(* IEC 61131-3 sources: std_i2980_v2.06_cp053/Source/IMM/ieccontrol/GlobalBaseArchives (part 2) *)

(* ---- ABVersionManager.pu ---- *)
(*
This algorithm block contains algorithms for version reading:
IEC and HMI version from version info text file
Firmware version from catalog
and stores them to sv_HMIVersion, sv_IECVersion and sv_FirmwareVersion
*)

IMPORT_OVER_LISTFILE
 KCAT_GetHandle
, KFILE_Open
, KFILE_Close
, tsTraceLevel
, KCAT_HandleData
, KCAT_Status
, KCAT_GenericDataFlags
, KCAT_RetCode

END_IMPORT

ALGORITHM_BLOCK ABVersionManager #DUMMY_EDIT_BLOCK

SYSTEM_VAR
 sv_TraceLevel : tsTraceLevel;
END_VAR

VAR
 msOsVersion : STRING(255);
 msDeviceSwVersion : STRING(255);
 msFirmwareVersion : STRING(255);
 msSystemName : STRING(255);
 msIECVersion : STRING(255);
 msCustVersion : STRING(255);
 msKVBVersion : STRING(255);
 msLIBIECBase : STRING(255);
 msLIBIECLib : STRING(255);
 msLIBException : STRING(255);
 msLIBODC : STRING(255);
END_VAR

FUNCTION fHasVersionInfoExtended : BOOL
 #DUMMY_EDIT_BLOCK
#BEGIN_EDIT_BLOCK

fHasVersionInfoExtended := (msDeviceSwVersion <> 'no version info' AND msOsVersion <> 'no version info');

;#END_EDIT_BLOCK END_FUNCTION

(*
This algo will copy the firmware version from the catalog entry to the sv_FirmwareVersion
*)

ALGORITHM aReadVersionInfo

VAR_INPUT
 sNodeName : STRING(255);
END_VAR

VAR_IN_OUT
 sVersionInfo : STRING(255);
END_VAR

VAR
 DataHandle : KCAT_HandleData;
 KCATStatus : KCAT_Status;
 dummy : DINT;
END_VAR
#BEGIN_EDIT_BLOCK
DataHandle := KCAT_GetHandle(sNodeName);
KCATStatus := DataHandle.Status;

IF (KCATStatus = KCAT_Status_OK) THEN
   KCATStatus := KCAT_GetValue(DataHandle.Handle, sVersionInfo);
END_IF;

IF ((KCATStatus <> KCAT_Status_OK) OR (sVersionInfo = '')) THEN
   sVersionInfo := "no version info";
   dummy := Print('Entry %s could not be found in catalog', sNodeName);
END_IF;

;#END_EDIT_BLOCK END_ALGORITHM

(*
This algo will copy the firmware version from the catalog entry to the sv_FirmwareVersion
*)

ALGORITHM aReadAllVersionInfos

VAR
 dummy : DINT;
END_VAR
#BEGIN_EDIT_BLOCK
aReadVersionInfo('System.firmwareVersion', msFirmwareVersion);
aReadVersionInfo('Application.KePlast.systemName', msSystemName);
aReadVersionInfo('Application.KePlast.IEC.componentVersionString', msIECVersion);
aReadVersionInfo('Application.KePlast.HMI.KVB.componentVersionString', msKVBVersion);

//aReadVersionInfo('Application.ApplMoldMachineKVBBase.componentVersionString', msLIBKVBBase);
aReadVersionInfo('Application.ApplIECUserExceptionHandling.componentVersionString', msLIBException);
aReadVersionInfo('Application.ApplMoldMachineIECLib.componentVersionString', msLIBIECLib);
aReadVersionInfo('Application.ApplMoldMachineIECBase.componentVersionString', msLIBIECBase);
aReadVersionInfo('Application.ApplMoldMachineODC.componentVersionString', msLIBODC);
aReadVersionInfo('BootVis.displayText', msCustVersion);
aReadVersionInfo('System.OS.driversVersion', msDeviceSwVersion);
aReadVersionInfo('System.OS.osVersion', msOsVersion);

IF (sv_TraceLevel.bApplication) THEN
   dummy := Print('ABVersionManager.aReadAllVersionInfos:');
   dummy := Print('  Version System:   "%s"', msSystemName);
   dummy := Print('  Version Firmware: "%s"', msFirmwareVersion);
   dummy := Print('  Version IEC:      "%s"', msIECVersion);
   dummy := Print('  Version KVB:      "%s"', msKVBVersion);
   dummy := Print('  Version IECLib:   "%s"', msLIBIECLib);
   dummy := Print('  Version IECBase:  "%s"', msLIBIECBase);
   dummy := Print('  Version Customer: "%s"', msCustVersion);
   IF (fHasVersionInfoExtended()) THEN
      dummy := Print('  Version DeviceSw: "%s"', msDeviceSwVersion);
      dummy := Print('  Version OS:       "%s"', msOsVersion);
   END_IF;
   dummy := Print('--------------------------------------');
END_IF;

;#END_EDIT_BLOCK END_ALGORITHM

FUNCTION fGetSystemName : STRING(255)
 #DUMMY_EDIT_BLOCK
#BEGIN_EDIT_BLOCK
fGetSystemName := msSystemName;

;#END_EDIT_BLOCK END_FUNCTION

FUNCTION fGetIECVersion : STRING(255)
 #DUMMY_EDIT_BLOCK
#BEGIN_EDIT_BLOCK
fGetIECVersion := msIECVersion;

;#END_EDIT_BLOCK END_FUNCTION

FUNCTION fGetCustVersion : STRING(255)
 #DUMMY_EDIT_BLOCK
#BEGIN_EDIT_BLOCK
fGetCustVersion := msCustVersion;

;#END_EDIT_BLOCK END_FUNCTION

FUNCTION fGetLIBVersionIECBase : STRING(255)
 #DUMMY_EDIT_BLOCK
#BEGIN_EDIT_BLOCK
fGetLIBVersionIECBase := msLIBIECBase;

;#END_EDIT_BLOCK END_FUNCTION

FUNCTION fGetLIBVersionIECLib : STRING(255)
 #DUMMY_EDIT_BLOCK
#BEGIN_EDIT_BLOCK
fGetLIBVersionIECLib := msLIBIECLib;

;#END_EDIT_BLOCK END_FUNCTION

FUNCTION fGetLIBVersionIECException : STRING(255)
 #DUMMY_EDIT_BLOCK
#BEGIN_EDIT_BLOCK
fGetLIBVersionIECException := msLIBException;

;#END_EDIT_BLOCK END_FUNCTION

FUNCTION fGetKVBVersion : STRING(255)
 #DUMMY_EDIT_BLOCK
#BEGIN_EDIT_BLOCK
fGetKVBVersion := msKVBVersion;

;#END_EDIT_BLOCK END_FUNCTION

(*
read KVS version on each function call because it never will be available at startup of IEC
*)

FUNCTION fReadKVSVersion : STRING(255)
 #DUMMY_EDIT_BLOCK

VAR
 sKVSVersion : STRING(255);
END_VAR
#BEGIN_EDIT_BLOCK
aReadVersionInfo('Application.KePlast.HMI.KVS.componentVersionString', sKVSVersion);
fReadKVSVersion := sKVSVersion;

;#END_EDIT_BLOCK END_FUNCTION

FUNCTION fGetFirmwareVersion : STRING(255)
 #DUMMY_EDIT_BLOCK
#BEGIN_EDIT_BLOCK
fGetFirmwareVersion := msFirmwareVersion;

;#END_EDIT_BLOCK END_FUNCTION

FUNCTION fGetLIBVersionODC : STRING(255)
 #DUMMY_EDIT_BLOCK
#BEGIN_EDIT_BLOCK
fGetLIBVersionODC := msLIBODC;

;#END_EDIT_BLOCK END_FUNCTION

FUNCTION fGetCPUSerial : LINT
 #DUMMY_EDIT_BLOCK

VAR
 sSerialNumber : STRING(255);
 flags : KCAT_GenericDataFlags;
 catRetCode : KCAT_RetCode;
 catHdl : KCAT_HandleData;
END_VAR
#BEGIN_EDIT_BLOCK
// get cpu serial number
catHdl := KCAT_GetHandle('IO.ONBOARD');
IF (catHdl.Status = KCAT_Status_OK) THEN
   catRetCode := KCAT_GetGenericData(catHdl.Handle, KCAT_GDSelector_SerialNumber, flags, sSerialNumber);
   IF (catRetCode = 0) THEN
      fGetCPUSerial := STRING_TO_LINT(sSerialNumber);
   END_IF;
END_IF;

;#END_EDIT_BLOCK END_FUNCTION

FUNCTION fGetDeviceSoftwareVersion : STRING(255)
 #DUMMY_EDIT_BLOCK
#BEGIN_EDIT_BLOCK
fGetDeviceSoftwareVersion := msDeviceSwVersion;

;#END_EDIT_BLOCK END_FUNCTION

FUNCTION fGetOSVersion : STRING(255)
 #DUMMY_EDIT_BLOCK
#BEGIN_EDIT_BLOCK
fGetOSVersion := msOsVersion;

;#END_EDIT_BLOCK END_FUNCTION

END_ALGORITHM_BLOCK

#END_OF_IEC_PART

@Puma @IecEditor 6 97 @Pou 25
@@@BEG_Comment@@@
This algorithm block contains algorithms for version reading:
IEC and HMI version from version info text file
Firmware version from catalog
and stores them to sv_HMIVersion, sv_IECVersion and sv_FirmwareVersion
@@@END_Comment@@@

@BEG_Contents

@BEG_Func
@RT(17)FuncTreeContainer
3
@Var @RT(14)KCAT_GetHandle @RT(0) @T @T @DERIVED 0 @F @RT(22)KEBA_STANDARD_FUNCTION @F
@T
@BEG_Attrib
0 @RT(0) @RT(0)
@END_Attrib
1 1 @F @F @F @F

@Var @RT(10)KFILE_Open @RT(0) @T @T @DERIVED 0 @F @RT(22)KEBA_STANDARD_FUNCTION @F
@T
@BEG_Attrib
0 @RT(0) @RT(0)
@END_Attrib
1 1 @F @F @F @F

@Var @RT(11)KFILE_Close @RT(0) @T @T @DERIVED 0 @F @RT(22)KEBA_STANDARD_FUNCTION @F
@T
@BEG_Attrib
0 @RT(0) @RT(0)
@END_Attrib
1 1 @F @F @F @F

@END_Func

@BEG_Const
@RT(18)ConstTreeContainer
0
@END_Const

@BEG_Export

@BEG_Kind
@ALGORITHM_BLOCK @RT(16)ABVersionManager @STRUCTURED_TEXT
@RT(0) @RT(0) @RT(0)
@END_Kind

@BEG_Dcl
@RT(16)DclTreeContainer
12
@Var @RT(13)sv_TraceLevel @RT(0) @T @T @DERIVED 0 @T @T @DT @RT(12)tsTraceLevel @RT(0) @T @T @UNKNOWN 0 @F
@F @F
@T
@BEG_Attrib
3 @RT(0) @RT(0) @RT(0)
@END_Attrib
1 8 @F @F @F @F

@Var @RT(11)msOsVersion @RT(0) @T @F @DT @RT(11)STRING(255) @RT(0) @T @T @STRING 0 @F @RT(3)255 @F
@F @F
@T
@BEG_Attrib
3 @RT(0) @RT(0) @RT(0)
@END_Attrib
1 0 @F @F @F @F

@Var @RT(17)msDeviceSwVersion @RT(0) @T @F @DT @RT(11)STRING(255) @RT(0) @T @T @STRING 0 @F @RT(3)255 @F
@F @F
@T
@BEG_Attrib
3 @RT(0) @RT(0) @RT(0)
@END_Attrib
1 0 @F @F @F @F

@Var @RT(17)msFirmwareVersion @RT(0) @T @F @DT @RT(11)STRING(255) @RT(0) @T @T @STRING 0 @F @RT(3)255 @F
@F @F
@T
@BEG_Attrib
3 @RT(0) @RT(0) @RT(0)
@END_Attrib
1 0 @F @F @F @F

@Var @RT(12)msSystemName @RT(0) @T @F @DT @RT(11)STRING(255) @RT(0) @T @T @STRING 0 @F @RT(3)255 @F
@F @F
@T
@BEG_Attrib
3 @RT(0) @RT(0) @RT(0)
@END_Attrib
1 0 @F @F @F @F

@Var @RT(12)msIECVersion @RT(0) @T @F @DT @RT(11)STRING(255) @RT(0) @T @T @STRING 0 @F @RT(3)255 @F
@F @F
@T
@BEG_Attrib
3 @RT(0) @RT(0) @RT(0)
@END_Attrib
1 0 @F @F @F @F

@Var @RT(13)msCustVersion @RT(0) @T @F @DT @RT(11)STRING(255) @RT(0) @T @T @STRING 0 @F @RT(3)255 @F
@F @F
@T
@BEG_Attrib
3 @RT(0) @RT(0) @RT(0)
@END_Attrib
1 0 @F @F @F @F

@Var @RT(12)msKVBVersion @RT(0) @T @F @DT @RT(11)STRING(255) @RT(0) @T @T @STRING 0 @F @RT(3)255 @F
@F @F
@T
@BEG_Attrib
3 @RT(0) @RT(0) @RT(0)
@END_Attrib
1 0 @F @F @F @F

@Var @RT(12)msLIBIECBase @RT(0) @T @F @DT @RT(11)STRING(255) @RT(0) @T @T @STRING 0 @F @RT(3)255 @F
@F @F
@T
@BEG_Attrib
3 @RT(0) @RT(0) @RT(0)
@END_Attrib
1 0 @F @F @F @F

@Var @RT(11)msLIBIECLib @RT(0) @T @F @DT @RT(11)STRING(255) @RT(0) @T @T @STRING 0 @F @RT(3)255 @F
@F @F
@T
@BEG_Attrib
3 @RT(0) @RT(0) @RT(0)
@END_Attrib
1 0 @F @F @F @F

@Var @RT(14)msLIBException @RT(0) @T @F @DT @RT(11)STRING(255) @RT(0) @T @T @STRING 0 @F @RT(3)255 @F
@F @F
@T
@BEG_Attrib
3 @RT(0) @RT(0) @RT(0)
@END_Attrib
1 0 @F @F @F @F

@Var @RT(8)msLIBODC @RT(0) @T @F @DT @RT(11)STRING(255) @RT(0) @T @T @STRING 0 @F @RT(3)255 @F
@F @F
@T
@BEG_Attrib
3 @RT(0) @RT(0) @RT(0)
@END_Attrib
1 0 @F @F @F @F

@END_Dcl

@END_Export

@BEG_Body

16

@BEG_Export

@BEG_Algo
@FUNCTION @RT(23)fHasVersionInfoExtended @STRUCTURED_TEXT
@RT(4)BOOL @RT(0) @RT(0) @F @F
@END_Algo

@BEG_Dcl
@RT(16)DclTreeContainer
0
@END_Dcl

@END_Export

@BEG_Export

@BEG_Algo
@ALGORITHM @RT(16)aReadVersionInfo @STRUCTURED_TEXT
@RT(0) @RT(0) @RT(0) @F @F
@END_Algo

@BEG_Dcl
@RT(16)DclTreeContainer
5
@Var @RT(10)DataHandle @RT(0) @T @T @DERIVED 0 @T @T @DT @RT(15)KCAT_HandleData @RT(0) @T @T @UNKNOWN 0 @F
@F @F
@T
@BEG_Attrib
3 @RT(0) @RT(0) @RT(0)
@END_Attrib
1 0 @F @F @F @F

@Var @RT(10)KCATStatus @RT(0) @T @T @DERIVED 0 @T @T @DT @RT(11)KCAT_Status @RT(0) @T @T @UNKNOWN 0 @F
@F @F
@T
@BEG_Attrib
3 @RT(0) @RT(0) @RT(0)
@END_Attrib
1 0 @F @F @F @F

@Var @RT(5)dummy @RT(0) @T @F @DT @RT(4)DINT @RT(0) @T @T @BASIC 0 @F
@F @F
@T
@BEG_Attrib
3 @RT(0) @RT(0) @RT(0)
@END_Attrib
1 0 @F @F @F @F

@Var @RT(9)sNodeName @RT(0) @T @F @DT @RT(11)STRING(255) @RT(0) @T @T @STRING 0 @F @RT(3)255 @F
@F @F
@T
@BEG_Attrib
3 @RT(0) @RT(0) @RT(0)
@END_Attrib
1 1 @F @F @F @F

@Var @RT(12)sVersionInfo @RT(0) @T @F @DT @RT(11)STRING(255) @RT(0) @T @T @STRING 0 @F @RT(3)255 @F
@F @F
@T
@BEG_Attrib
3 @RT(0) @RT(0) @RT(0)
@END_Attrib
1 2 @F @F @F @F

@END_Dcl

@END_Export

@BEG_Export

@BEG_Algo
@ALGORITHM @RT(20)aReadAllVersionInfos @STRUCTURED_TEXT
@RT(0) @RT(0) @RT(0) @F @F
@END_Algo

@BEG_Dcl
@RT(16)DclTreeContainer
1
@Var @RT(5)dummy @RT(0) @T @F @DT @RT(4)DINT @RT(0) @T @T @BASIC 0 @F
@F @F
@T
@BEG_Attrib
3 @RT(0) @RT(0) @RT(0)
@END_Attrib
1 0 @F @F @F @F

@END_Dcl

@END_Export

@BEG_Export

@BEG_Algo
@FUNCTION @RT(14)fGetSystemName @STRUCTURED_TEXT
@RT(11)STRING(255) @RT(0) @RT(0) @F @F
@END_Algo

@BEG_Dcl
@RT(16)DclTreeContainer
0
@END_Dcl

@END_Export

@BEG_Export

@BEG_Algo
@FUNCTION @RT(14)fGetIECVersion @STRUCTURED_TEXT
@RT(11)STRING(255) @RT(0) @RT(0) @F @F
@END_Algo

@BEG_Dcl
@RT(16)DclTreeContainer
0
@END_Dcl

@END_Export

@BEG_Export

@BEG_Algo
@FUNCTION @RT(15)fGetCustVersion @STRUCTURED_TEXT
@RT(11)STRING(255) @RT(0) @RT(0) @F @F
@END_Algo

@BEG_Dcl
@RT(16)DclTreeContainer
0
@END_Dcl

@END_Export

@BEG_Export

@BEG_Algo
@FUNCTION @RT(21)fGetLIBVersionIECBase @STRUCTURED_TEXT
@RT(11)STRING(255) @RT(0) @RT(0) @F @F
@END_Algo

@BEG_Dcl
@RT(16)DclTreeContainer
0
@END_Dcl

@END_Export

@BEG_Export

@BEG_Algo
@FUNCTION @RT(20)fGetLIBVersionIECLib @STRUCTURED_TEXT
@RT(11)STRING(255) @RT(0) @RT(0) @F @F
@END_Algo

@BEG_Dcl
@RT(16)DclTreeContainer
0
@END_Dcl

@END_Export

@BEG_Export

@BEG_Algo
@FUNCTION @RT(26)fGetLIBVersionIECException @STRUCTURED_TEXT
@RT(11)STRING(255) @RT(0) @RT(0) @F @F
@END_Algo

@BEG_Dcl
@RT(16)DclTreeContainer
0
@END_Dcl

@END_Export

@BEG_Export

@BEG_Algo
@FUNCTION @RT(14)fGetKVBVersion @STRUCTURED_TEXT
@RT(11)STRING(255) @RT(0) @RT(0) @F @F
@END_Algo

@BEG_Dcl
@RT(16)DclTreeContainer
0
@END_Dcl

@END_Export

@BEG_Export

@BEG_Algo
@FUNCTION @RT(15)fReadKVSVersion @STRUCTURED_TEXT
@RT(11)STRING(255) @RT(0) @RT(0) @F @F
@END_Algo

@BEG_Dcl
@RT(16)DclTreeContainer
1
@Var @RT(11)sKVSVersion @RT(0) @T @F @DT @RT(11)STRING(255) @RT(0) @T @T @STRING 0 @F @RT(3)255 @F
@F @F
@T
@BEG_Attrib
3 @RT(0) @RT(0) @RT(0)
@END_Attrib
1 0 @F @F @F @F

@END_Dcl

@END_Export

@BEG_Export

@BEG_Algo
@FUNCTION @RT(19)fGetFirmwareVersion @STRUCTURED_TEXT
@RT(11)STRING(255) @RT(0) @RT(0) @F @F
@END_Algo

@BEG_Dcl
@RT(16)DclTreeContainer
0
@END_Dcl

@END_Export

@BEG_Export

@BEG_Algo
@FUNCTION @RT(17)fGetLIBVersionODC @STRUCTURED_TEXT
@RT(11)STRING(255) @RT(0) @RT(0) @F @F
@END_Algo

@BEG_Dcl
@RT(16)DclTreeContainer
0
@END_Dcl

@END_Export

@BEG_Export

@BEG_Algo
@FUNCTION @RT(13)fGetCPUSerial @STRUCTURED_TEXT
@RT(4)LINT @RT(0) @RT(0) @F @F
@END_Algo

@BEG_Dcl
@RT(16)DclTreeContainer
4
@Var @RT(13)sSerialNumber @RT(0) @T @F @DT @RT(11)STRING(255) @RT(0) @T @T @STRING 0 @F @RT(3)255 @F
@F @F
@T
@BEG_Attrib
3 @RT(0) @RT(0) @RT(0)
@END_Attrib
1 0 @F @F @F @F

@Var @RT(5)flags @RT(0) @T @T @DERIVED 0 @T @T @DT @RT(21)KCAT_GenericDataFlags @RT(0) @T @T @UNKNOWN 0 @F
@F @F
@T
@BEG_Attrib
3 @RT(0) @RT(0) @RT(0)
@END_Attrib
1 0 @F @F @F @F

@Var @RT(10)catRetCode @RT(0) @T @T @DERIVED 0 @T @T @DT @RT(12)KCAT_RetCode @RT(0) @T @T @UNKNOWN 0 @F
@F @F
@T
@BEG_Attrib
3 @RT(0) @RT(0) @RT(0)
@END_Attrib
1 0 @F @F @F @F

@Var @RT(6)catHdl @RT(0) @T @T @DERIVED 0 @T @T @DT @RT(15)KCAT_HandleData @RT(0) @T @T @UNKNOWN 0 @F
@F @F
@T
@BEG_Attrib
3 @RT(0) @RT(0) @RT(0)
@END_Attrib
1 0 @F @F @F @F

@END_Dcl

@END_Export

@BEG_Export

@BEG_Algo
@FUNCTION @RT(25)fGetDeviceSoftwareVersion @STRUCTURED_TEXT
@RT(11)STRING(255) @RT(0) @RT(0) @F @F
@END_Algo

@BEG_Dcl
@RT(16)DclTreeContainer
0
@END_Dcl

@END_Export

@BEG_Export

@BEG_Algo
@FUNCTION @RT(13)fGetOSVersion @STRUCTURED_TEXT
@RT(11)STRING(255) @RT(0) @RT(0) @F @F
@END_Algo

@BEG_Dcl
@RT(16)DclTreeContainer
0
@END_Dcl

@END_Export

@BEG_Body
@TL(3)

fHasVersionInfoExtended := (msDeviceSwVersion <> 'no version info' AND msOsVersion <> 'no version info');

@END_Body

@@@BEG_Comment@@@
@TL(0)

@@@END_Comment@@@

@BEG_Body
@TL(12)
DataHandle := KCAT_GetHandle(sNodeName);
KCATStatus := DataHandle.Status;

IF (KCATStatus = KCAT_Status_OK) THEN
   KCATStatus := KCAT_GetValue(DataHandle.Handle, sVersionInfo);
END_IF;

IF ((KCATStatus <> KCAT_Status_OK) OR (sVersionInfo = '')) THEN
   sVersionInfo := "no version info";
   dummy := Print('Entry %s could not be found in catalog', sNodeName);
END_IF;

@END_Body

@@@BEG_Comment@@@
@TL(1)
This algo will copy the firmware version from the catalog entry to the sv_FirmwareVersion
@@@END_Comment@@@

@BEG_Body
@TL(30)
aReadVersionInfo('System.firmwareVersion', msFirmwareVersion);
aReadVersionInfo('Application.KePlast.systemName', msSystemName);
aReadVersionInfo('Application.KePlast.IEC.componentVersionString', msIECVersion);
aReadVersionInfo('Application.KePlast.HMI.KVB.componentVersionString', msKVBVersion);

//aReadVersionInfo('Application.ApplMoldMachineKVBBase.componentVersionString', msLIBKVBBase);
aReadVersionInfo('Application.ApplIECUserExceptionHandling.componentVersionString', msLIBException);
aReadVersionInfo('Application.ApplMoldMachineIECLib.componentVersionString', msLIBIECLib);
aReadVersionInfo('Application.ApplMoldMachineIECBase.componentVersionString', msLIBIECBase);
aReadVersionInfo('Application.ApplMoldMachineODC.componentVersionString', msLIBODC);
aReadVersionInfo('BootVis.displayText', msCustVersion);
aReadVersionInfo('System.OS.driversVersion', msDeviceSwVersion);
aReadVersionInfo('System.OS.osVersion', msOsVersion);

IF (sv_TraceLevel.bApplication) THEN
   dummy := Print('ABVersionManager.aReadAllVersionInfos:');
   dummy := Print('  Version System:   "%s"', msSystemName);
   dummy := Print('  Version Firmware: "%s"', msFirmwareVersion);
   dummy := Print('  Version IEC:      "%s"', msIECVersion);
   dummy := Print('  Version KVB:      "%s"', msKVBVersion);
   dummy := Print('  Version IECLib:   "%s"', msLIBIECLib);
   dummy := Print('  Version IECBase:  "%s"', msLIBIECBase);
   dummy := Print('  Version Customer: "%s"', msCustVersion);
   IF (fHasVersionInfoExtended()) THEN
      dummy := Print('  Version DeviceSw: "%s"', msDeviceSwVersion);
      dummy := Print('  Version OS:       "%s"', msOsVersion);
   END_IF;
   dummy := Print('--------------------------------------');
END_IF;

@END_Body

@@@BEG_Comment@@@
@TL(1)
This algo will copy the firmware version from the catalog entry to the sv_FirmwareVersion
@@@END_Comment@@@

@BEG_Body
@TL(2)
fGetSystemName := msSystemName;

@END_Body

@@@BEG_Comment@@@
@TL(0)

@@@END_Comment@@@

@BEG_Body
@TL(2)
fGetIECVersion := msIECVersion;

@END_Body

@@@BEG_Comment@@@
@TL(0)

@@@END_Comment@@@

@BEG_Body
@TL(2)
fGetCustVersion := msCustVersion;

@END_Body

@@@BEG_Comment@@@
@TL(0)

@@@END_Comment@@@

@BEG_Body
@TL(2)
fGetLIBVersionIECBase := msLIBIECBase;

@END_Body

@@@BEG_Comment@@@
@TL(0)

@@@END_Comment@@@

@BEG_Body
@TL(2)
fGetLIBVersionIECLib := msLIBIECLib;

@END_Body

@@@BEG_Comment@@@
@TL(0)

@@@END_Comment@@@

@BEG_Body
@TL(2)
fGetLIBVersionIECException := msLIBException;

@END_Body

@@@BEG_Comment@@@
@TL(0)

@@@END_Comment@@@

@BEG_Body
@TL(2)
fGetKVBVersion := msKVBVersion;

@END_Body

@@@BEG_Comment@@@
@TL(0)

@@@END_Comment@@@

@BEG_Body
@TL(3)
aReadVersionInfo('Application.KePlast.HMI.KVS.componentVersionString', sKVSVersion);
fReadKVSVersion := sKVSVersion;

@END_Body

@@@BEG_Comment@@@
@TL(1)
read KVS version on each function call because it never will be available at startup of IEC
@@@END_Comment@@@

@BEG_Body
@TL(2)
fGetFirmwareVersion := msFirmwareVersion;

@END_Body

@@@BEG_Comment@@@
@TL(0)

@@@END_Comment@@@

@BEG_Body
@TL(2)
fGetLIBVersionODC := msLIBODC;

@END_Body

@@@BEG_Comment@@@
@TL(0)

@@@END_Comment@@@

@BEG_Body
@TL(10)
// get cpu serial number
catHdl := KCAT_GetHandle('IO.ONBOARD');
IF (catHdl.Status = KCAT_Status_OK) THEN
   catRetCode := KCAT_GetGenericData(catHdl.Handle, KCAT_GDSelector_SerialNumber, flags, sSerialNumber);
   IF (catRetCode = 0) THEN
      fGetCPUSerial := STRING_TO_LINT(sSerialNumber);
   END_IF;
END_IF;

@END_Body

@@@BEG_Comment@@@
@TL(0)

@@@END_Comment@@@

@BEG_Body
@TL(3)
fGetDeviceSoftwareVersion := msDeviceSwVersion;

@END_Body

@@@BEG_Comment@@@
@TL(0)

@@@END_Comment@@@

@BEG_Body
@TL(3)
fGetOSVersion := msOsVersion;

@END_Body

@@@BEG_Comment@@@
@TL(0)

@@@END_Comment@@@
@END_Body

@END_Contents

(* ---- ASSERT.pu ---- *)
(*
@h    ! WARNING !
@h    The Kemro K2 system (including software) only meets category B according to EN 954-1,
@h    thus it is not intended for usage in safety-relevant control applications in the field
@h    of personal safety (e.g. emergency stop).
@h    To implement potentially necessary safety-relevant control tasks, always use additional
@h    external safety devices that are intended for the particular purpose, and meet the necessary
@h    functional safety.
@h    For further information see EN 954-1 (EN ISO 13849-1) and/or the K2-x00 user manual, chapter
@h    "CE conformity, directives and standards".

*)

IMPORT_OVER_LISTFILE
 STOP_SYSTEM
, SET_ALARM
, KSYS_Status
, KCAT_Status
, KCAT_HandleData

END_IMPORT

FUNCTION ASSERT : BOOL #DUMMY_EDIT_BLOCK

VAR_INPUT
 b : BOOL;
 erAssert : ALARM;
END_VAR

VAR
 dummy : DINT;
 Status : KSYS_Status;
 StatusCat : KCAT_Status;
 DataHandle : KCAT_HandleData;
 iLogEnable : DINT;
END_VAR

VAR CONSTANT
 iNull : DINT := 0;
END_VAR
#BEGIN_EDIT_BLOCK
(**************************************** WARNING ********************************************
 *** The KEBA Kemro K2 System including software is not intended for safety control tasks! ***
 ***                       For further information see Comment tab!                        ***
 *********************************************************************************************)

ASSERT := b;

IF b THEN
    RETURN;
END_IF;

dummy := Print('$n$n$n');
dummy := Print('************************************************************');
dummy := Print('***************** KePlast.IEC: ASSERT **********************');
dummy := Print('******************** stopping system ***********************');
dummy := Print('************************************************************$n$n$n');

DataHandle := KCAT_GetHandle('System.LogEnable');
IF DataHandle.Status = KCAT_Status_OK THEN
   StatusCat := KCAT_GetValue(Handle := DataHandle.Handle,
   Buffer := iLogEnable);
END_IF;

SET_ALARM(erAssert);

IF iLogEnable = 1 THEN
    Status:=SET_WVEVENT(9999);
END_IF;

dummy := dummy / iNull;

STOP_SYSTEM();

;#END_EDIT_BLOCK END_FUNCTION

#END_OF_IEC_PART

@Puma @IecEditor 6 96 @Pou 25
@@@BEG_Comment@@@
@h    ! WARNING !
@h    The Kemro K2 system (including software) only meets category B according to EN 954-1,
@h    thus it is not intended for usage in safety-relevant control applications in the field
@h    of personal safety (e.g. emergency stop).
@h    To implement potentially necessary safety-relevant control tasks, always use additional
@h    external safety devices that are intended for the particular purpose, and meet the necessary
@h    functional safety.
@h    For further information see EN 954-1 (EN ISO 13849-1) and/or the K2-x00 user manual, chapter
@h    "CE conformity, directives and standards".

@@@END_Comment@@@

@BEG_Contents

@BEG_Func
@RT(17)FuncTreeContainer
2
@Var @RT(11)STOP_SYSTEM @RT(0) @T @T @DERIVED 0 @F @RT(23)KEBA_STANDARD_PROCEDURE @F
@T
@BEG_Attrib
0 @RT(0) @RT(0)
@END_Attrib
1 1 @F @F @F @F

@Var @RT(9)SET_ALARM @RT(0) @T @T @DERIVED 0 @F @RT(23)KEBA_STANDARD_PROCEDURE @F
@T
@BEG_Attrib
0 @RT(0) @RT(0)
@END_Attrib
1 1 @F @F @F @F

@END_Func

@BEG_Const
@RT(18)ConstTreeContainer
0
@END_Const

@BEG_Export

@BEG_Kind
@FUNCTION @RT(6)ASSERT @STRUCTURED_TEXT
@RT(4)BOOL @RT(0) @RT(0)
@END_Kind

@BEG_Dcl
@RT(16)DclTreeContainer
8
@Var @RT(5)dummy @RT(0) @T @F @DT @RT(4)DINT @RT(0) @T @T @BASIC 0 @F
@F @F
@T
@BEG_Attrib
3 @RT(0) @RT(0) @RT(0)
@END_Attrib
1 0 @F @F @F @F

@Var @RT(1)b @RT(0) @T @F @DT @RT(4)BOOL @RT(0) @T @T @BASIC 0 @F
@F @F
@T
@BEG_Attrib
3 @RT(0) @RT(0) @RT(0)
@END_Attrib
1 1 @F @F @F @F

@Var @RT(5)iNull @RT(0) @T @F @DT @RT(4)DINT @RT(0) @T @T @BASIC 0 @F
@F @F
@T
@BEG_Attrib
3 @RT(1)0 @RT(0) @RT(0)
@END_Attrib
1 15 @F @F @F @F

@Var @RT(8)erAssert @RT(0) @T @F @DT @RT(5)ALARM @RT(0) @T @T @BASIC 0 @F
@F @F
@T
@BEG_Attrib
3 @RT(0) @RT(0) @RT(0)
@END_Attrib
1 1 @F @F @F @F

@Var @RT(6)Status @RT(0) @T @T @DERIVED 0 @T @T @DT @RT(11)KSYS_Status @RT(0) @T @T @UNKNOWN 0 @F
@F @F
@T
@BEG_Attrib
3 @RT(0) @RT(0) @RT(0)
@END_Attrib
1 0 @F @F @F @F

@Var @RT(9)StatusCat @RT(0) @T @T @DERIVED 0 @F @RT(11)KCAT_Status @F
@T
@BEG_Attrib
3 @RT(0) @RT(0) @RT(0)
@END_Attrib
1 0 @F @F @F @F

@Var @RT(10)DataHandle @RT(0) @T @T @DERIVED 0 @F @RT(15)KCAT_HandleData @F
@T
@BEG_Attrib
3 @RT(0) @RT(0) @RT(0)
@END_Attrib
1 0 @F @F @F @F

@Var @RT(10)iLogEnable @RT(0) @T @F @DT @RT(4)DINT @RT(0) @T @T @BASIC 0 @F
@F @F
@T
@BEG_Attrib
3 @RT(0) @RT(0) @RT(0)
@END_Attrib
1 0 @F @F @F @F

@END_Dcl

@END_Export

@BEG_Body
@TL(34)
(**************************************** WARNING ********************************************
 *** The KEBA Kemro K2 System including software is not intended for safety control tasks! ***
 ***                       For further information see Comment tab!                        ***
 *********************************************************************************************)

ASSERT := b;

IF b THEN
    RETURN;
END_IF;

dummy := Print('$n$n$n');
dummy := Print('************************************************************');
dummy := Print('***************** KePlast.IEC: ASSERT **********************');
dummy := Print('******************** stopping system ***********************');
dummy := Print('************************************************************$n$n$n');

DataHandle := KCAT_GetHandle('System.LogEnable');
IF DataHandle.Status = KCAT_Status_OK THEN
   StatusCat := KCAT_GetValue(Handle := DataHandle.Handle,
   Buffer := iLogEnable);
END_IF;

SET_ALARM(erAssert);

IF iLogEnable = 1 THEN
    Status:=SET_WVEVENT(9999);
END_IF;

dummy := dummy / iNull;

STOP_SYSTEM();

@END_Body

@END_Contents

(* ---- FCalcDuration.pu ---- *)
IMPORT_OVER_LISTFILE
 KCTRL_Prof_Light

END_IMPORT

FUNCTION FCalcDuration : TIME #DUMMY_EDIT_BLOCK

VAR_INPUT
 StartPosition : REAL (* start position of actual movement *);
 StartVelocity : REAL (* start velocity of actual movement *);
 EndPosition : REAL (* end position of actual movement *);
 Profile : KCTRL_Prof_Light (* calculated profile for non constant movement *);
 StartRamp : REAL (* start ramp for all movements *);
 StopRamp : REAL (* stop ramp for interposition or constant movement *);
 ConstOutput : REAL (* constant velocity *);
 UseConstOutput : BOOL (* movement with constant velocity *);
END_VAR

VAR
 bDir : BOOL;
 iStartIndex : UDINT;
 iEndIndex : UDINT;
 iActIndex : UDINT;
 rDuration : REAL;
 rEndVelocity : REAL;
 rEndVelocityStart : REAL;
 rCuttingPosition : REAL;
 rCuttingPositionEnd : REAL;
 rAcceleration : REAL;
 rDeltaPosStart : REAL;
 rDeltaPosStop : REAL;
 rDeltaT1 : REAL;
 rDeltaT2 : REAL;
 rDeltaT3 : REAL;
 rStopRamp : REAL;
 rPositionDifference : REAL;
 rStartVelocity : REAL;
END_VAR

VAR CONSTANT
 cMaxDuration : REAL := 1.0e10;
END_VAR
#BEGIN_EDIT_BLOCK
rDuration := 0.0;

IF UseConstOutput THEN

    //Constant movement
    IF ConstOutput <= 0.0 THEN
        FCalcDuration := T#0s;
        RETURN;
    END_IF;
    IF StartRamp > 0.0 THEN
        rDeltaPosStart := 0.5 * ConstOutput*ConstOutput / StartRamp;
        rDeltaT3 := ConstOutput / StartRamp;
    ELSE
        FCalcDuration := T#0s;
        RETURN;
    END_IF;
    IF StopRamp > 0.0 THEN
        rDeltaPosStop := 0.5 * ConstOutput*ConstOutput / StopRamp;
        rDeltaT3 := ConstOutput / StopRamp;
    ELSE
        rDeltaPosStop := 0.0;
        rDeltaT3 := 0.0;
    END_IF;
    IF (rDeltaPosStop + rDeltaPosStart) < ABS(EndPosition - StartPosition) THEN
        rDeltaT2 := (ABS(EndPosition - StartPosition) - rDeltaPosStop - rDeltaPosStart) / ConstOutput;
    ELSE
        IF ((StartRamp*StopRamp) > 0.0) THEN
            rDeltaT1 := SQRT(2.0 * ABS(EndPosition - StartPosition) * StopRamp / StartRamp /(StartRamp + StopRamp));
            rDeltaT3 := SQRT(2.0 * ABS(EndPosition - StartPosition) * StartRamp / StopRamp /(StartRamp + StopRamp));
        ELSE
            rDeltaT1 := 0.0;
            rDeltaT3 := 0.0;
        END_IF;
        rDeltaT2 := 0.0;
    END_IF;

ELSE
    IF StartRamp <= 0.0 THEN
        FCalcDuration := T#0s;
        RETURN;
    END_IF;
    IF StopRamp <= 0.0 THEN
        rStopRamp := StartRamp;
    ELSE
        rStopRamp := StopRamp;
    END_IF;
    IF StartVelocity  < 0.0 THEN
        rStartVelocity := 0.0;
    ELSE
        rStartVelocity := StartVelocity;
    END_IF;

    //Profile movement
    IF (Profile.uNoOfPoints > 0) THEN
        IF (Profile.Point[Profile.uNoOfPoints].rX > Profile.Point[1].rX) THEN
            bDir := TRUE;
        ELSIF (Profile.Point[Profile.uNoOfPoints].rX < Profile.Point[1].rX) THEN
            bDir := FALSE;
        ELSE // only one point
            IF (Profile.Point[Profile.uNoOfPoints].rY > 0.0) THEN
                rDuration := ABS((StartPosition - EndPosition) / Profile.Point[Profile.uNoOfPoints].rY);
                IF (rDuration > cMaxDuration) OR (rDuration < 0.0) THEN
                    rDuration := 0.0;
                END_IF;
                FCalcDuration := LINT_TO_TIME(REAL_TO_LINT(rDuration*1.0e6));
            ELSE
                FCalcDuration := T#0s;
            END_IF;
            RETURN;
        END_IF;
        // no movement necessary
        IF ((bDir      AND (StartPosition >= EndPosition))OR
           ((NOT bDir) AND (StartPosition <= EndPosition))) THEN
            FCalcDuration := T#0s;
            RETURN;
        END_IF;
        // end point not in profile
        IF ((bDir      AND (Profile.Point[1].rX >= EndPosition))OR
           ((NOT bDir) AND (Profile.Point[1].rX <= EndPosition))) THEN
            FCalcDuration := T#0s;
            RETURN;
        END_IF;
    ELSE
        FCalcDuration := T#0s;
        RETURN;
    END_IF;

    // start ramp
    iActIndex := 0;
    iStartIndex := Profile.uNoOfPoints;
    rCuttingPosition := Profile.Point[iStartIndex].rX;
    WHILE (iActIndex < Profile.uNoOfPoints) DO
        iActIndex := iActIndex + 1;
        IF ((bDir      AND (StartPosition < Profile.Point[iActIndex].rX))OR
           ((NOT bDir) AND (StartPosition > Profile.Point[iActIndex].rX))) THEN
            rEndVelocity := SQRT(rStartVelocity*rStartVelocity +
                                2.0 * StartRamp * ABS(StartPosition - Profile.Point[iActIndex].rX));
            IF (rEndVelocity >= Profile.Point[iActIndex].rY) THEN
                iStartIndex := iActIndex;
                IF (iActIndex > 1) THEN
                    // avoid divide by "0" if jumps in profile allowed/calculated
                    IF (Profile.Point[iActIndex].rX = Profile.Point[iActIndex-1].rX) THEN
                        rCuttingPosition := Profile.Point[iActIndex].rX;
                    ELSE
                        rAcceleration := ((Profile.Point[iActIndex].rY * Profile.Point[iActIndex].rY) -
                                          (Profile.Point[iActIndex-1].rY * Profile.Point[iActIndex-1].rY)) /
                                       ABS(Profile.Point[iActIndex].rX - Profile.Point[iActIndex-1].rX);
                        IF (bDir) THEN
                            //xEnd = (x_0 + a*p[j].y*p[j].y - a*p[j].x*fact) /((float)1.0-a*fact);
                            rCuttingPosition := (StartPosition +
                                                 Profile.Point[iStartIndex].rY*Profile.Point[iStartIndex].rY*0.5/StartRamp -
                                                 Profile.Point[iStartIndex].rX*rAcceleration*0.5/StartRamp)/
                                                (1.0-0.5*rAcceleration/StartRamp);
                        ELSE
                            //xEnd = (x_0 - a*p[j].y*p[j].y - a*p[j].x*fact) /((float)1.0-a*fact);
                            rCuttingPosition := (StartPosition -
                                                 Profile.Point[iStartIndex].rY*Profile.Point[iStartIndex].rY*0.5/StartRamp -
                                                 Profile.Point[iStartIndex].rX*rAcceleration*0.5/StartRamp)/
                                                (1.0-0.5*rAcceleration/StartRamp);
                        END_IF;
                    END_IF;
                ELSE
                   IF (bDir) THEN
                        //xEnd = (x_0 + a*p[j].y*p[j].y - a*p[j].x*fact) /((float)1.0-a*fact);
                        rCuttingPosition := (StartPosition + Profile.Point[iStartIndex].rY*Profile.Point[iStartIndex].rY*0.5/StartRamp);
                    ELSE
                        //xEnd = (x_0 - a*p[j].y*p[j].y - a*p[j].x*fact) /((float)1.0-a*fact);
                        rCuttingPosition := (StartPosition - Profile.Point[iStartIndex].rY*Profile.Point[iStartIndex].rY*0.5/StartRamp);
                    END_IF;
                    rDuration := 0.0;
                END_IF;
                EXIT;
            END_IF;
        END_IF;
    END_WHILE;

    // stop ramp
    iActIndex := 0;
    iEndIndex := 1;
    rCuttingPositionEnd := EndPosition;
    IF ((bDir      AND (EndPosition >= Profile.Point[Profile.uNoOfPoints].rX))OR
       ((NOT bDir) AND (EndPosition <= Profile.Point[Profile.uNoOfPoints].rX))) THEN
        rCuttingPositionEnd := EndPosition;//Profile.Point[Profile.uNoOfPoints].rX;
        iEndIndex := Profile.uNoOfPoints;
    ELSE
        iActIndex := Profile.uNoOfPoints;
        WHILE (iActIndex > 1) DO
            iActIndex := iActIndex - 1;
            IF ((bDir      AND (EndPosition >= Profile.Point[iActIndex].rX))OR
               ((NOT bDir) AND (EndPosition <= Profile.Point[iActIndex].rX))) THEN
                rEndVelocity := SQRT(rStartVelocity*rStartVelocity +
                    2.0 * rStopRamp * ABS(EndPosition - Profile.Point[iActIndex].rX));

                IF (rEndVelocity >= Profile.Point[iActIndex].rY) THEN
                    iEndIndex := iActIndex;
                    // avoid divide by "0" if jumps in profile allowed/calculated
                    IF (Profile.Point[iActIndex+1].rX = Profile.Point[iActIndex].rX) THEN
                        rCuttingPositionEnd := EndPosition;
                    ELSE
                        rAcceleration := ((Profile.Point[iActIndex+1].rY * Profile.Point[iActIndex+1].rY) -
                                          (Profile.Point[iActIndex].rY * Profile.Point[iActIndex].rY)) /
                                       ABS(Profile.Point[iActIndex+1].rX - Profile.Point[iActIndex].rX);
                        IF (ABS(2.0*rStopRamp+rAcceleration) > 0.0) THEN
                            IF (bDir) THEN
                                // xCut = xEnd - (yStart*yStart - 2*aProfil*xStart)/(2*aStop+aProfil)
                                rCuttingPositionEnd := EndPosition -
                                                      (Profile.Point[iEndIndex].rY*Profile.Point[iEndIndex].rY +
                                                      (EndPosition - Profile.Point[iEndIndex].rX)*rAcceleration)/
                                                      (2.0*rStopRamp+rAcceleration);
                            ELSE
                                // xCut = xEnd + (yStart*yStart - 2*aProfil*xStart)/(2*aStop+aProfil)
                                rCuttingPositionEnd := EndPosition +
                                                      (Profile.Point[iEndIndex].rY*Profile.Point[iEndIndex].rY +
                                                      (Profile.Point[iEndIndex].rX - EndPosition)*rAcceleration)/
                                                      (2.0*rStopRamp+rAcceleration);
                            END_IF;
                        ELSE
                            rCuttingPositionEnd := Profile.Point[iEndIndex].rX;
                        END_IF;
                    END_IF;
                    EXIT;
                ELSE
                    IF (iActIndex = 1) THEN
                        IF (bDir) THEN
                            rCuttingPositionEnd := EndPosition -
                                Profile.Point[1].rY * Profile.Point[1].rY * 0.5 / rStopRamp;
                        ELSE
                            rCuttingPositionEnd := EndPosition +
                                Profile.Point[1].rY * Profile.Point[1].rY * 0.5 / rStopRamp;
                        END_IF;
                        EXIT;
                    END_IF;
                END_IF;
            END_IF;

        END_WHILE;
    END_IF;

    // add up times
    IF ((bDir      AND (rCuttingPositionEnd >= rCuttingPosition))OR
       ((NOT bDir) AND (rCuttingPositionEnd <= rCuttingPosition))) THEN

        // start ramp
        rEndVelocityStart := SQRT(rStartVelocity*rStartVelocity +
                            2.0 *ABS(StartPosition - rCuttingPosition) * StartRamp);
        IF ((rStartVelocity + rEndVelocityStart) > 0.0) THEN
            rDeltaT1 := 2.0 * ABS((StartPosition - rCuttingPosition) /
                                                (rStartVelocity + rEndVelocityStart));
            IF (iStartIndex <= iEndIndex) THEN
                rDeltaT1 :=  rDeltaT1 +
                    2.0 * ABS((Profile.Point[iStartIndex].rX - rCuttingPosition) /
                    (Profile.Point[iStartIndex].rY + rEndVelocityStart));
            END_IF;
        ELSE
            rDeltaT1 := 0.0;
        END_IF;

        // stop ramp        iEndIndex := Profile.uNoOfPoints;
        rEndVelocity := SQRT(2.0 *ABS(EndPosition - rCuttingPositionEnd) * rStopRamp);
        IF (rEndVelocity > 0.0) THEN
            rDeltaT2 := 2.0 * ABS((EndPosition - rCuttingPositionEnd) / rEndVelocity);
            IF (iEndIndex >= iStartIndex) THEN
                rDeltaT2 :=  rDeltaT2 +
                    2.0 * ABS((Profile.Point[iEndIndex].rX - rCuttingPositionEnd) /
                    (Profile.Point[iEndIndex].rY + rEndVelocity));
            ELSE
                rDeltaT2 :=  rDeltaT2 +
                    2.0 * ABS((rCuttingPosition - rCuttingPositionEnd) /
                    (rEndVelocityStart + rEndVelocity));
            END_IF;
        ELSE
            rDeltaT2 := 0.0;
        END_IF;

        // steps between start and stop
        rDeltaT3 := 0.0;
        FOR iActIndex:= iStartIndex+1 TO iEndIndex DO
            IF ((Profile.Point[iActIndex].rY + Profile.Point[iActIndex-1].rY) > 0.0) THEN
                rDeltaT3 := rDeltaT3 + 2.0 * ABS(
                            (Profile.Point[iActIndex].rX - Profile.Point[iActIndex-1].rX)/
                            (Profile.Point[iActIndex].rY + Profile.Point[iActIndex-1].rY));
            END_IF;
        END_FOR;
    ELSE //  only start ramp and stop ramp
        // calc intersection point of two ramps
        rPositionDifference := ABS(StartPosition - EndPosition);
        rCuttingPosition := (rStopRamp* rPositionDifference - 0.5 * rStartVelocity*rStartVelocity)/(StartRamp + rStopRamp);
        IF (rCuttingPosition > 0.0) THEN // position difference > 0 -> end velocity > 0
            rEndVelocity := SQRT(rStartVelocity*rStartVelocity + 2.0 * rCuttingPosition * StartRamp);
            rDuration := 2.0 * ((rPositionDifference - rCuttingPosition)/ rEndVelocity + rCuttingPosition /(rEndVelocity + rStartVelocity));
        ELSE
            IF rStartVelocity > 0.0 THEN
               rDuration := 2.0 * rPositionDifference / rStartVelocity;
            ELSE
               rDuration := 0.0;
            END_IF;
        END_IF;
        IF (rDuration > cMaxDuration) OR (rDuration < 0.0) THEN
            rDuration := 0.0;
        END_IF;
        FCalcDuration := LINT_TO_TIME(REAL_TO_LINT(rDuration*1.0e6));
        RETURN;
    END_IF;

END_IF;

rDuration := rDeltaT1 + rDeltaT2 + rDeltaT3;
IF (rDuration > cMaxDuration) OR (rDuration < 0.0) THEN
    rDuration := 0.0;
END_IF;
FCalcDuration := LINT_TO_TIME(REAL_TO_LINT(rDuration*1.0e6));

;#END_EDIT_BLOCK END_FUNCTION

#END_OF_IEC_PART

@Puma @IecEditor 6 131 @Pou 25
@@@BEG_Comment@@@

@@@END_Comment@@@

@BEG_Contents

@BEG_Func
@RT(17)FuncTreeContainer
0
@END_Func

@BEG_Const
@RT(18)ConstTreeContainer
0
@END_Const

@BEG_Export

@BEG_Kind
@FUNCTION @RT(13)FCalcDuration @STRUCTURED_TEXT
@RT(4)TIME @RT(0) @RT(0)
@END_Kind

@BEG_Dcl
@RT(16)DclTreeContainer
27
@Var @RT(13)StartPosition @RT(0) @T @F @DT @RT(4)REAL @RT(0) @T @T @BASIC 0 @F
@F @F
@T
@BEG_Attrib
3 @RT(0) @RT(33)start position of actual movement @RT(0)
@END_Attrib
1 1 @F @F @F @F

@Var @RT(13)StartVelocity @RT(0) @T @F @DT @RT(4)REAL @RT(0) @T @T @BASIC 0 @F
@F @F
@T
@BEG_Attrib
3 @RT(0) @RT(33)start velocity of actual movement @RT(0)
@END_Attrib
1 1 @F @F @F @F

@Var @RT(11)EndPosition @RT(0) @T @F @DT @RT(4)REAL @RT(0) @T @T @BASIC 0 @F
@F @F
@T
@BEG_Attrib
3 @RT(0) @RT(31)end position of actual movement @RT(0)
@END_Attrib
1 1 @F @F @F @F

@Var @RT(7)Profile @RT(0) @T @T @DERIVED 0 @T @T @DT @RT(16)KCTRL_Prof_Light @RT(0) @T @T @UNKNOWN 0 @F
@F @F
@T
@BEG_Attrib
3 @RT(0) @RT(44)calculated profile for non constant movement @RT(0)
@END_Attrib
1 1 @F @F @F @F

@Var @RT(9)StartRamp @RT(0) @T @F @DT @RT(4)REAL @RT(0) @T @T @BASIC 0 @F
@F @F
@T
@BEG_Attrib
3 @RT(0) @RT(28)start ramp for all movements @RT(0)
@END_Attrib
1 1 @F @F @F @F

@Var @RT(8)StopRamp @RT(0) @T @F @DT @RT(4)REAL @RT(0) @T @T @BASIC 0 @F
@F @F
@T
@BEG_Attrib
3 @RT(0) @RT(48)stop ramp for interposition or constant movement @RT(0)
@END_Attrib
1 1 @F @F @F @F

@Var @RT(11)ConstOutput @RT(0) @T @F @DT @RT(4)REAL @RT(0) @T @T @BASIC 0 @F
@F @F
@T
@BEG_Attrib
3 @RT(0) @RT(17)constant velocity @RT(0)
@END_Attrib
1 1 @F @F @F @F

@Var @RT(14)UseConstOutput @RT(0) @T @F @DT @RT(4)BOOL @RT(0) @T @T @BASIC 0 @F
@F @F
@T
@BEG_Attrib
3 @RT(0) @RT(31)movement with constant velocity @RT(0)
@END_Attrib
1 1 @F @F @F @F

@Var @RT(4)bDir @RT(0) @T @F @DT @RT(4)BOOL @RT(0) @T @T @BASIC 0 @F
@F @F
@T
@BEG_Attrib
3 @RT(0) @RT(0) @RT(0)
@END_Attrib
1 0 @F @F @F @F

@Var @RT(11)iStartIndex @RT(0) @T @F @DT @RT(5)UDINT @RT(0) @T @T @BASIC 0 @F
@F @F
@T
@BEG_Attrib
3 @RT(0) @RT(0) @RT(0)
@END_Attrib
1 0 @F @F @F @F

@Var @RT(9)iEndIndex @RT(0) @T @F @DT @RT(5)UDINT @RT(0) @T @T @BASIC 0 @F
@F @F
@T
@BEG_Attrib
3 @RT(0) @RT(0) @RT(0)
@END_Attrib
1 0 @F @F @F @F

@Var @RT(9)iActIndex @RT(0) @T @F @DT @RT(5)UDINT @RT(0) @T @T @BASIC 0 @F
@F @F
@T
@BEG_Attrib
3 @RT(0) @RT(0) @RT(0)
@END_Attrib
1 0 @F @F @F @F

@Var @RT(9)rDuration @RT(0) @T @F @DT @RT(4)REAL @RT(0) @T @T @BASIC 0 @F
@F @F
@T
@BEG_Attrib
3 @RT(0) @RT(0) @RT(0)
@END_Attrib
1 0 @F @F @F @F

@Var @RT(12)rEndVelocity @RT(0) @T @F @DT @RT(4)REAL @RT(0) @T @T @BASIC 0 @F
@F @F
@T
@BEG_Attrib
3 @RT(0) @RT(0) @RT(0)
@END_Attrib
1 0 @F @F @F @F

@Var @RT(17)rEndVelocityStart @RT(0) @T @F @DT @RT(4)REAL @RT(0) @T @T @BASIC 0 @F
@F @F
@T
@BEG_Attrib
3 @RT(0) @RT(0) @RT(0)
@END_Attrib
1 0 @F @F @F @F

@Var @RT(16)rCuttingPosition @RT(0) @T @F @DT @RT(4)REAL @RT(0) @T @T @BASIC 0 @F
@F @F
@T
@BEG_Attrib
3 @RT(0) @RT(0) @RT(0)
@END_Attrib
1 0 @F @F @F @F

@Var @RT(19)rCuttingPositionEnd @RT(0) @T @F @DT @RT(4)REAL @RT(0) @T @T @BASIC 0 @F
@F @F
@T
@BEG_Attrib
3 @RT(0) @RT(0) @RT(0)
@END_Attrib
1 0 @F @F @F @F

@Var @RT(13)rAcceleration @RT(0) @T @F @DT @RT(4)REAL @RT(0) @T @T @BASIC 0 @F
@F @F
@T
@BEG_Attrib
3 @RT(0) @RT(0) @RT(0)
@END_Attrib
1 0 @F @F @F @F

@Var @RT(14)rDeltaPosStart @RT(0) @T @F @DT @RT(4)REAL @RT(0) @T @T @BASIC 0 @F
@F @F
@T
@BEG_Attrib
3 @RT(0) @RT(0) @RT(0)
@END_Attrib
1 0 @F @F @F @F

@Var @RT(13)rDeltaPosStop @RT(0) @T @F @DT @RT(4)REAL @RT(0) @T @T @BASIC 0 @F
@F @F
@T
@BEG_Attrib
3 @RT(0) @RT(0) @RT(0)
@END_Attrib
1 0 @F @F @F @F

@Var @RT(8)rDeltaT1 @RT(0) @T @F @DT @RT(4)REAL @RT(0) @T @T @BASIC 0 @F
@F @F
@T
@BEG_Attrib
3 @RT(0) @RT(0) @RT(0)
@END_Attrib
1 0 @F @F @F @F

@Var @RT(8)rDeltaT2 @RT(0) @T @F @DT @RT(4)REAL @RT(0) @T @T @BASIC 0 @F
@F @F
@T
@BEG_Attrib
3 @RT(0) @RT(0) @RT(0)
@END_Attrib
1 0 @F @F @F @F

@Var @RT(8)rDeltaT3 @RT(0) @T @F @DT @RT(4)REAL @RT(0) @T @T @BASIC 0 @F
@F @F
@T
@BEG_Attrib
3 @RT(0) @RT(0) @RT(0)
@END_Attrib
1 0 @F @F @F @F

@Var @RT(9)rStopRamp @RT(0) @T @F @DT @RT(4)REAL @RT(0) @T @T @BASIC 0 @F
@F @F
@T
@BEG_Attrib
3 @RT(0) @RT(0) @RT(0)
@END_Attrib
1 0 @F @F @F @F

@Var @RT(19)rPositionDifference @RT(0) @T @F @DT @RT(4)REAL @RT(0) @T @T @BASIC 0 @F
@F @F
@T
@BEG_Attrib
3 @RT(0) @RT(0) @RT(0)
@END_Attrib
1 0 @F @F @F @F

@Var @RT(14)rStartVelocity @RT(0) @T @F @DT @RT(4)REAL @RT(0) @T @T @BASIC 0 @F
@F @F
@T
@BEG_Attrib
3 @RT(0) @RT(0) @RT(0)
@END_Attrib
1 0 @F @F @F @F

@Var @RT(12)cMaxDuration @RT(0) @T @F @DT @RT(4)REAL @RT(0) @T @T @BASIC 0 @F
@F @F
@T
@BEG_Attrib
3 @RT(6)1.0e10 @RT(0) @RT(0)
@END_Attrib
1 15 @F @F @F @F

@END_Dcl

@END_Export

@BEG_Body
@TL(273)
rDuration := 0.0;

IF UseConstOutput THEN

    //Constant movement
    IF ConstOutput <= 0.0 THEN
        FCalcDuration := T#0s;
        RETURN;
    END_IF;
    IF StartRamp > 0.0 THEN
        rDeltaPosStart := 0.5 * ConstOutput*ConstOutput / StartRamp;
        rDeltaT3 := ConstOutput / StartRamp;
    ELSE
        FCalcDuration := T#0s;
        RETURN;
    END_IF;
    IF StopRamp > 0.0 THEN
        rDeltaPosStop := 0.5 * ConstOutput*ConstOutput / StopRamp;
        rDeltaT3 := ConstOutput / StopRamp;
    ELSE
        rDeltaPosStop := 0.0;
        rDeltaT3 := 0.0;
    END_IF;
    IF (rDeltaPosStop + rDeltaPosStart) < ABS(EndPosition - StartPosition) THEN
        rDeltaT2 := (ABS(EndPosition - StartPosition) - rDeltaPosStop - rDeltaPosStart) / ConstOutput;
    ELSE
        IF ((StartRamp*StopRamp) > 0.0) THEN
            rDeltaT1 := SQRT(2.0 * ABS(EndPosition - StartPosition) * StopRamp / StartRamp /(StartRamp + StopRamp));
            rDeltaT3 := SQRT(2.0 * ABS(EndPosition - StartPosition) * StartRamp / StopRamp /(StartRamp + StopRamp));
        ELSE
            rDeltaT1 := 0.0;
            rDeltaT3 := 0.0;
        END_IF;
        rDeltaT2 := 0.0;
    END_IF;

ELSE
    IF StartRamp <= 0.0 THEN
        FCalcDuration := T#0s;
        RETURN;
    END_IF;
    IF StopRamp <= 0.0 THEN
        rStopRamp := StartRamp;
    ELSE
        rStopRamp := StopRamp;
    END_IF;
    IF StartVelocity  < 0.0 THEN
        rStartVelocity := 0.0;
    ELSE
        rStartVelocity := StartVelocity;
    END_IF;

    //Profile movement
    IF (Profile.uNoOfPoints > 0) THEN
        IF (Profile.Point[Profile.uNoOfPoints].rX > Profile.Point[1].rX) THEN
            bDir := TRUE;
        ELSIF (Profile.Point[Profile.uNoOfPoints].rX < Profile.Point[1].rX) THEN
            bDir := FALSE;
        ELSE // only one point
            IF (Profile.Point[Profile.uNoOfPoints].rY > 0.0) THEN
                rDuration := ABS((StartPosition - EndPosition) / Profile.Point[Profile.uNoOfPoints].rY);
                IF (rDuration > cMaxDuration) OR (rDuration < 0.0) THEN
                    rDuration := 0.0;
                END_IF;
                FCalcDuration := LINT_TO_TIME(REAL_TO_LINT(rDuration*1.0e6));
            ELSE
                FCalcDuration := T#0s;
            END_IF;
            RETURN;
        END_IF;
        // no movement necessary
        IF ((bDir      AND (StartPosition >= EndPosition))OR
           ((NOT bDir) AND (StartPosition <= EndPosition))) THEN
            FCalcDuration := T#0s;
            RETURN;
        END_IF;
        // end point not in profile
        IF ((bDir      AND (Profile.Point[1].rX >= EndPosition))OR
           ((NOT bDir) AND (Profile.Point[1].rX <= EndPosition))) THEN
            FCalcDuration := T#0s;
            RETURN;
        END_IF;
    ELSE
        FCalcDuration := T#0s;
        RETURN;
    END_IF;

    // start ramp
    iActIndex := 0;
    iStartIndex := Profile.uNoOfPoints;
    rCuttingPosition := Profile.Point[iStartIndex].rX;
    WHILE (iActIndex < Profile.uNoOfPoints) DO
        iActIndex := iActIndex + 1;
        IF ((bDir      AND (StartPosition < Profile.Point[iActIndex].rX))OR
           ((NOT bDir) AND (StartPosition > Profile.Point[iActIndex].rX))) THEN
            rEndVelocity := SQRT(rStartVelocity*rStartVelocity +
                                2.0 * StartRamp * ABS(StartPosition - Profile.Point[iActIndex].rX));
            IF (rEndVelocity >= Profile.Point[iActIndex].rY) THEN
                iStartIndex := iActIndex;
                IF (iActIndex > 1) THEN
                    // avoid divide by "0" if jumps in profile allowed/calculated
                    IF (Profile.Point[iActIndex].rX = Profile.Point[iActIndex-1].rX) THEN
                        rCuttingPosition := Profile.Point[iActIndex].rX;
                    ELSE
                        rAcceleration := ((Profile.Point[iActIndex].rY * Profile.Point[iActIndex].rY) -
                                          (Profile.Point[iActIndex-1].rY * Profile.Point[iActIndex-1].rY)) /
                                       ABS(Profile.Point[iActIndex].rX - Profile.Point[iActIndex-1].rX);
                        IF (bDir) THEN
                            //xEnd = (x_0 + a*p[j].y*p[j].y - a*p[j].x*fact) /((float)1.0-a*fact);
                            rCuttingPosition := (StartPosition +
                                                 Profile.Point[iStartIndex].rY*Profile.Point[iStartIndex].rY*0.5/StartRamp -
                                                 Profile.Point[iStartIndex].rX*rAcceleration*0.5/StartRamp)/
                                                (1.0-0.5*rAcceleration/StartRamp);
                        ELSE
                            //xEnd = (x_0 - a*p[j].y*p[j].y - a*p[j].x*fact) /((float)1.0-a*fact);
                            rCuttingPosition := (StartPosition -
                                                 Profile.Point[iStartIndex].rY*Profile.Point[iStartIndex].rY*0.5/StartRamp -
                                                 Profile.Point[iStartIndex].rX*rAcceleration*0.5/StartRamp)/
                                                (1.0-0.5*rAcceleration/StartRamp);
                        END_IF;
                    END_IF;
                ELSE
                   IF (bDir) THEN
                        //xEnd = (x_0 + a*p[j].y*p[j].y - a*p[j].x*fact) /((float)1.0-a*fact);
                        rCuttingPosition := (StartPosition + Profile.Point[iStartIndex].rY*Profile.Point[iStartIndex].rY*0.5/StartRamp);
                    ELSE
                        //xEnd = (x_0 - a*p[j].y*p[j].y - a*p[j].x*fact) /((float)1.0-a*fact);
                        rCuttingPosition := (StartPosition - Profile.Point[iStartIndex].rY*Profile.Point[iStartIndex].rY*0.5/StartRamp);
                    END_IF;
                    rDuration := 0.0;
                END_IF;
                EXIT;
            END_IF;
        END_IF;
    END_WHILE;

    // stop ramp
    iActIndex := 0;
    iEndIndex := 1;
    rCuttingPositionEnd := EndPosition;
    IF ((bDir      AND (EndPosition >= Profile.Point[Profile.uNoOfPoints].rX))OR
       ((NOT bDir) AND (EndPosition <= Profile.Point[Profile.uNoOfPoints].rX))) THEN
        rCuttingPositionEnd := EndPosition;//Profile.Point[Profile.uNoOfPoints].rX;
        iEndIndex := Profile.uNoOfPoints;
    ELSE
        iActIndex := Profile.uNoOfPoints;
        WHILE (iActIndex > 1) DO
            iActIndex := iActIndex - 1;
            IF ((bDir      AND (EndPosition >= Profile.Point[iActIndex].rX))OR
               ((NOT bDir) AND (EndPosition <= Profile.Point[iActIndex].rX))) THEN
                rEndVelocity := SQRT(rStartVelocity*rStartVelocity +
                    2.0 * rStopRamp * ABS(EndPosition - Profile.Point[iActIndex].rX));

                IF (rEndVelocity >= Profile.Point[iActIndex].rY) THEN
                    iEndIndex := iActIndex;
                    // avoid divide by "0" if jumps in profile allowed/calculated
                    IF (Profile.Point[iActIndex+1].rX = Profile.Point[iActIndex].rX) THEN
                        rCuttingPositionEnd := EndPosition;
                    ELSE
                        rAcceleration := ((Profile.Point[iActIndex+1].rY * Profile.Point[iActIndex+1].rY) -
                                          (Profile.Point[iActIndex].rY * Profile.Point[iActIndex].rY)) /
                                       ABS(Profile.Point[iActIndex+1].rX - Profile.Point[iActIndex].rX);
                        IF (ABS(2.0*rStopRamp+rAcceleration) > 0.0) THEN
                            IF (bDir) THEN
                                // xCut = xEnd - (yStart*yStart - 2*aProfil*xStart)/(2*aStop+aProfil)
                                rCuttingPositionEnd := EndPosition -
                                                      (Profile.Point[iEndIndex].rY*Profile.Point[iEndIndex].rY +
                                                      (EndPosition - Profile.Point[iEndIndex].rX)*rAcceleration)/
                                                      (2.0*rStopRamp+rAcceleration);
                            ELSE
                                // xCut = xEnd + (yStart*yStart - 2*aProfil*xStart)/(2*aStop+aProfil)
                                rCuttingPositionEnd := EndPosition +
                                                      (Profile.Point[iEndIndex].rY*Profile.Point[iEndIndex].rY +
                                                      (Profile.Point[iEndIndex].rX - EndPosition)*rAcceleration)/
                                                      (2.0*rStopRamp+rAcceleration);
                            END_IF;
                        ELSE
                            rCuttingPositionEnd := Profile.Point[iEndIndex].rX;
                        END_IF;
                    END_IF;
                    EXIT;
                ELSE
                    IF (iActIndex = 1) THEN
                        IF (bDir) THEN
                            rCuttingPositionEnd := EndPosition -
                                Profile.Point[1].rY * Profile.Point[1].rY * 0.5 / rStopRamp;
                        ELSE
                            rCuttingPositionEnd := EndPosition +
                                Profile.Point[1].rY * Profile.Point[1].rY * 0.5 / rStopRamp;
                        END_IF;
                        EXIT;
                    END_IF;
                END_IF;
            END_IF;

        END_WHILE;
    END_IF;

    // add up times
    IF ((bDir      AND (rCuttingPositionEnd >= rCuttingPosition))OR
       ((NOT bDir) AND (rCuttingPositionEnd <= rCuttingPosition))) THEN

        // start ramp
        rEndVelocityStart := SQRT(rStartVelocity*rStartVelocity +
                            2.0 *ABS(StartPosition - rCuttingPosition) * StartRamp);
        IF ((rStartVelocity + rEndVelocityStart) > 0.0) THEN
            rDeltaT1 := 2.0 * ABS((StartPosition - rCuttingPosition) /
                                                (rStartVelocity + rEndVelocityStart));
            IF (iStartIndex <= iEndIndex) THEN
                rDeltaT1 :=  rDeltaT1 +
                    2.0 * ABS((Profile.Point[iStartIndex].rX - rCuttingPosition) /
                    (Profile.Point[iStartIndex].rY + rEndVelocityStart));
            END_IF;
        ELSE
            rDeltaT1 := 0.0;
        END_IF;

        // stop ramp        iEndIndex := Profile.uNoOfPoints;
        rEndVelocity := SQRT(2.0 *ABS(EndPosition - rCuttingPositionEnd) * rStopRamp);
        IF (rEndVelocity > 0.0) THEN
            rDeltaT2 := 2.0 * ABS((EndPosition - rCuttingPositionEnd) / rEndVelocity);
            IF (iEndIndex >= iStartIndex) THEN
                rDeltaT2 :=  rDeltaT2 +
                    2.0 * ABS((Profile.Point[iEndIndex].rX - rCuttingPositionEnd) /
                    (Profile.Point[iEndIndex].rY + rEndVelocity));
            ELSE
                rDeltaT2 :=  rDeltaT2 +
                    2.0 * ABS((rCuttingPosition - rCuttingPositionEnd) /
                    (rEndVelocityStart + rEndVelocity));
            END_IF;
        ELSE
            rDeltaT2 := 0.0;
        END_IF;

        // steps between start and stop
        rDeltaT3 := 0.0;
        FOR iActIndex:= iStartIndex+1 TO iEndIndex DO
            IF ((Profile.Point[iActIndex].rY + Profile.Point[iActIndex-1].rY) > 0.0) THEN
                rDeltaT3 := rDeltaT3 + 2.0 * ABS(
                            (Profile.Point[iActIndex].rX - Profile.Point[iActIndex-1].rX)/
                            (Profile.Point[iActIndex].rY + Profile.Point[iActIndex-1].rY));
            END_IF;
        END_FOR;
    ELSE //  only start ramp and stop ramp
        // calc intersection point of two ramps
        rPositionDifference := ABS(StartPosition - EndPosition);
        rCuttingPosition := (rStopRamp* rPositionDifference - 0.5 * rStartVelocity*rStartVelocity)/(StartRamp + rStopRamp);
        IF (rCuttingPosition > 0.0) THEN // position difference > 0 -> end velocity > 0
            rEndVelocity := SQRT(rStartVelocity*rStartVelocity + 2.0 * rCuttingPosition * StartRamp);
            rDuration := 2.0 * ((rPositionDifference - rCuttingPosition)/ rEndVelocity + rCuttingPosition /(rEndVelocity + rStartVelocity));
        ELSE
            IF rStartVelocity > 0.0 THEN
               rDuration := 2.0 * rPositionDifference / rStartVelocity;
            ELSE
               rDuration := 0.0;
            END_IF;
        END_IF;
        IF (rDuration > cMaxDuration) OR (rDuration < 0.0) THEN
            rDuration := 0.0;
        END_IF;
        FCalcDuration := LINT_TO_TIME(REAL_TO_LINT(rDuration*1.0e6));
        RETURN;
    END_IF;

END_IF;

rDuration := rDeltaT1 + rDeltaT2 + rDeltaT3;
IF (rDuration > cMaxDuration) OR (rDuration < 0.0) THEN
    rDuration := 0.0;
END_IF;
FCalcDuration := LINT_TO_TIME(REAL_TO_LINT(rDuration*1.0e6));

@END_Body

@END_Contents

(* ---- FCalcScrewCircumfenceSpeed.pu ---- *)
(*
calculate screw circumfence speed in cm/s
*)

FUNCTION FCalcScrewCircumfenceSpeed : REAL #DUMMY_EDIT_BLOCK

VAR_INPUT
 rDiameter : REAL;
 rRPM : REAL;
END_VAR

VAR CONSTANT
 PI : REAL := 3.14159265;
END_VAR
#BEGIN_EDIT_BLOCK
(**************************************** WARNING ********************************************
 *** The KEBA Kemro K2 System including software is not intended for safety control tasks! ***
 ***                       For further information see Comment tab!                        ***
 *********************************************************************************************)

FCalcScrewCircumfenceSpeed := rRPM / 60.0 * rDiameter * PI / 10.0;

;#END_EDIT_BLOCK END_FUNCTION

#END_OF_IEC_PART

@Puma @IecEditor 6 34 @Pou 25
@@@BEG_Comment@@@
calculate screw circumfence speed in cm/s
@@@END_Comment@@@

@BEG_Contents

@BEG_Func
@RT(17)FuncTreeContainer
0
@END_Func

@BEG_Const
@RT(18)ConstTreeContainer
0
@END_Const

@BEG_Export

@BEG_Kind
@FUNCTION @RT(26)FCalcScrewCircumfenceSpeed @STRUCTURED_TEXT
@RT(4)REAL @RT(0) @RT(0)
@END_Kind

@BEG_Dcl
@RT(16)DclTreeContainer
3
@Var @RT(9)rDiameter @RT(0) @T @F @DT @RT(4)REAL @RT(0) @T @T @BASIC 0 @F
@F @F
@T
@BEG_Attrib
3 @RT(0) @RT(0) @RT(0)
@END_Attrib
1 1 @F @F @F @F

@Var @RT(4)rRPM @RT(0) @T @F @DT @RT(4)REAL @RT(0) @T @T @BASIC 0 @F
@F @F
@T
@BEG_Attrib
3 @RT(0) @RT(0) @RT(0)
@END_Attrib
1 1 @F @F @F @F

@Var @RT(2)PI @RT(0) @T @F @DT @RT(4)REAL @RT(0) @T @T @BASIC 0 @F
@F @F
@T
@BEG_Attrib
3 @RT(10)3.14159265 @RT(0) @RT(0)
@END_Attrib
1 15 @F @F @F @F

@END_Dcl

@END_Export

@BEG_Body
@TL(9)
(**************************************** WARNING ********************************************
 *** The KEBA Kemro K2 System including software is not intended for safety control tasks! ***
 ***                       For further information see Comment tab!                        ***
 *********************************************************************************************)

FCalcScrewCircumfenceSpeed := rRPM / 60.0 * rDiameter * PI / 10.0;

@END_Body

@END_Contents

(* ---- FCalcScrewSize.pu ---- *)
(*
calculate screw plane in mm^2

*)

FUNCTION FCalcScrewSize : REAL #DUMMY_EDIT_BLOCK

VAR_INPUT
 rDiameter : REAL (* diameter of screw in mm *);
END_VAR

VAR CONSTANT
 PI : REAL := 3.14159265;
END_VAR
#BEGIN_EDIT_BLOCK
(**************************************** WARNING ********************************************
 *** The KEBA Kemro K2 System including software is not intended for safety control tasks! ***
 ***                       For further information see Comment tab!                        ***
 *********************************************************************************************)

(* calculate screw plane in mm^2 *)
FCalcScrewSize := EXPT(rDiameter, 2.0) * PI / 4.0

;#END_EDIT_BLOCK END_FUNCTION

#END_OF_IEC_PART

@Puma @IecEditor 6 30 @Pou 25
@@@BEG_Comment@@@
calculate screw plane in mm^2

@@@END_Comment@@@

@BEG_Contents

@BEG_Func
@RT(17)FuncTreeContainer
0
@END_Func

@BEG_Const
@RT(18)ConstTreeContainer
0
@END_Const

@BEG_Export

@BEG_Kind
@FUNCTION @RT(14)FCalcScrewSize @STRUCTURED_TEXT
@RT(4)REAL @RT(0) @RT(0)
@END_Kind

@BEG_Dcl
@RT(16)DclTreeContainer
2
@Var @RT(9)rDiameter @RT(0) @T @F @DT @RT(4)REAL @RT(0) @T @T @BASIC 0 @F
@F @F
@T
@BEG_Attrib
3 @RT(0) @RT(23)diameter of screw in mm @RT(0)
@END_Attrib
1 1 @F @F @F @F

@Var @RT(2)PI @RT(0) @T @F @DT @RT(4)REAL @RT(0) @T @T @BASIC 0 @F
@F @F
@T
@BEG_Attrib
3 @RT(10)3.14159265 @RT(0) @RT(0)
@END_Attrib
1 15 @F @F @F @F

@END_Dcl

@END_Export

@BEG_Body
@TL(8)
(**************************************** WARNING ********************************************
 *** The KEBA Kemro K2 System including software is not intended for safety control tasks! ***
 ***                       For further information see Comment tab!                        ***
 *********************************************************************************************)

(* calculate screw plane in mm^2 *)
FCalcScrewSize := EXPT(rDiameter, 2.0) * PI / 4.0

@END_Body

@END_Contents

(* ---- FCalcSetVelocity.pu ---- *)
FUNCTION FCalcSetVelocity : REAL #DUMMY_EDIT_BLOCK

VAR_INPUT
 rMaxVelocity : REAL (* max. velocity of movement *);
 rStroke : REAL (* max. stroke of movement *);
 dMaxMoveTime : TIME (* max. movetime *);
END_VAR

VAR
 rSetVelocity : REAL;
 rSetVelocityRel : REAL;
 rUsedStroke : REAL := 0.9 (* % of stroke used during movement *);
 rMaxVelocityRel : REAL := 99.0 (* % of max. velocity used during movement *);
END_VAR
#BEGIN_EDIT_BLOCK
rSetVelocity := rUsedStroke * rStroke / LINT_TO_REAL(TIME_TO_LINT(dMaxMoveTime)) * 1.0e6;
IF rMaxVelocity > 0.0 THEN
    IF rSetVelocity > rMaxVelocityRel / 100.0 * rMaxVelocity THEN
        rSetVelocity := rMaxVelocityRel / 100.0 * rMaxVelocity;
        rSetVelocityRel := rMaxVelocityRel;
    END_IF;
    rSetVelocityRel := rSetVelocity / rMaxVelocity * 100.0;
ELSE
    rSetVelocity := 0.0;
    rSetVelocityRel := 100.0;
END_IF;
FCalcSetVelocity := rSetVelocityRel;

;#END_EDIT_BLOCK END_FUNCTION

#END_OF_IEC_PART

@Puma @IecEditor 6 120 @Pou 25
@@@BEG_Comment@@@

@@@END_Comment@@@

@BEG_Contents

@BEG_Func
@RT(17)FuncTreeContainer
0
@END_Func

@BEG_Const
@RT(18)ConstTreeContainer
0
@END_Const

@BEG_Export

@BEG_Kind
@FUNCTION @RT(16)FCalcSetVelocity @STRUCTURED_TEXT
@RT(4)REAL @RT(0) @RT(0)
@END_Kind

@BEG_Dcl
@RT(16)DclTreeContainer
7
@Var @RT(12)rMaxVelocity @RT(0) @T @F @DT @RT(4)REAL @RT(0) @T @T @BASIC 0 @F
@F @F
@T
@BEG_Attrib
3 @RT(0) @RT(25)max. velocity of movement @RT(0)
@END_Attrib
1 1 @F @F @F @F

@Var @RT(7)rStroke @RT(0) @T @F @DT @RT(4)REAL @RT(0) @T @T @BASIC 0 @F
@F @F
@T
@BEG_Attrib
3 @RT(0) @RT(23)max. stroke of movement @RT(0)
@END_Attrib
1 1 @F @F @F @F

@Var @RT(12)dMaxMoveTime @RT(0) @T @F @DT @RT(4)TIME @RT(0) @T @T @BASIC 0 @F
@F @F
@T
@BEG_Attrib
3 @RT(0) @RT(13)max. movetime @RT(0)
@END_Attrib
1 1 @F @F @F @F

@Var @RT(12)rSetVelocity @RT(0) @T @F @DT @RT(4)REAL @RT(0) @T @T @BASIC 0 @F
@F @F
@T
@BEG_Attrib
3 @RT(0) @RT(0) @RT(0)
@END_Attrib
1 0 @F @F @F @F

@Var @RT(15)rSetVelocityRel @RT(0) @T @F @DT @RT(4)REAL @RT(0) @T @T @BASIC 0 @F
@F @F
@T
@BEG_Attrib
3 @RT(0) @RT(0) @RT(0)
@END_Attrib
1 0 @F @F @F @F

@Var @RT(11)rUsedStroke @RT(0) @T @F @DT @RT(4)REAL @RT(0) @T @T @BASIC 0 @F
@F @F
@T
@BEG_Attrib
3 @RT(3)0.9 @RT(32)% of stroke used during movement @RT(0)
@END_Attrib
1 0 @F @F @F @F

@Var @RT(15)rMaxVelocityRel @RT(0) @T @F @DT @RT(4)REAL @RT(0) @T @T @BASIC 0 @F
@F @F
@T
@BEG_Attrib
3 @RT(4)99.0 @RT(39)% of max. velocity used during movement @RT(0)
@END_Attrib
1 0 @F @F @F @F

@END_Dcl

@END_Export

@BEG_Body
@TL(13)
rSetVelocity := rUsedStroke * rStroke / LINT_TO_REAL(TIME_TO_LINT(dMaxMoveTime)) * 1.0e6;
IF rMaxVelocity > 0.0 THEN
    IF rSetVelocity > rMaxVelocityRel / 100.0 * rMaxVelocity THEN
        rSetVelocity := rMaxVelocityRel / 100.0 * rMaxVelocity;
        rSetVelocityRel := rMaxVelocityRel;
    END_IF;
    rSetVelocityRel := rSetVelocity / rMaxVelocity * 100.0;
ELSE
    rSetVelocity := 0.0;
    rSetVelocityRel := 100.0;
END_IF;
FCalcSetVelocity := rSetVelocityRel;

@END_Body

@END_Contents

(* ---- FCalculateCylinderSize.pu ---- *)
(*
calculate size of cylinder in mm^2
if bSmallSize is TRUE the size only includes the outer ring
*)

IMPORT_OVER_LISTFILE
 tsCylinderData

END_IMPORT

FUNCTION FCalculateCylinderSize : REAL #DUMMY_EDIT_BLOCK

VAR_INPUT
 CylinderData : tsCylinderData (* cylinder to calculate size from *);
 bSmallSize : BOOL (* subtract piston rod from size *);
 bCalcHighPressSize : BOOL;
END_VAR

VAR CONSTANT
 PI : REAL := 3.14159265;
END_VAR
#BEGIN_EDIT_BLOCK
(**************************************** WARNING ********************************************
 *** The KEBA Kemro K2 System including software is not intended for safety control tasks! ***
 ***                       For further information see Comment tab!                        ***
 *********************************************************************************************)

IF CylinderData.rPlungerDiameter <> 0.0 THEN  //plunger available
    IF CylinderData.bMoveWithPlunger THEN //plunger inside highpressure-cylinder -> only used for mold close
        IF bCalcHighPressSize THEN
            FCalculateCylinderSize := DINT_TO_REAL(CylinderData.iNumCylinders) *
                                        ((EXPT(CylinderData.rCylinderDiameter, 2.0) * PI / 4.0)-
                                        (EXPT(CylinderData.rPlungerDiameter, 2.0) * PI / 4.0));
        ELSE
            IF bSmallSize THEN
                FCalculateCylinderSize := DINT_TO_REAL(CylinderData.iNumCylinders) *
                                            ((EXPT(CylinderData.rCylinderDiameter, 2.0) * PI / 4.0)-
                                            (EXPT(CylinderData.rPistonRodDiameter, 2.0) * PI / 4.0));
            ELSE
                FCalculateCylinderSize := DINT_TO_REAL(CylinderData.iNumCylinders) *
                                            (EXPT(CylinderData.rPlungerDiameter, 2.0) * PI / 4.0);
            END_IF;
        END_IF;
    ELSE //plunger used for high pressure build up, differential cylinders used for mold movement
        IF bCalcHighPressSize THEN
            FCalculateCylinderSize := DINT_TO_REAL(CylinderData.iNumCylinders) *
                                        (EXPT(CylinderData.rPlungerDiameter, 2.0) * PI / 4.0);
        ELSE
            IF bSmallSize THEN
                FCalculateCylinderSize := DINT_TO_REAL(CylinderData.iNumCylinders) *
                                            ((EXPT(CylinderData.rCylinderDiameter, 2.0) * PI / 4.0)-
                                            (EXPT(CylinderData.rPistonRodDiameter, 2.0) * PI / 4.0));
            ELSE
                FCalculateCylinderSize := DINT_TO_REAL(CylinderData.iNumCylinders) *
                                            (EXPT(CylinderData.rCylinderDiameter, 2.0) * PI / 4.0);
            END_IF;
        END_IF;
    END_IF;
ELSE //no plunger
    IF bSmallSize THEN
        FCalculateCylinderSize := DINT_TO_REAL(CylinderData.iNumCylinders) *
                                    ((EXPT(CylinderData.rCylinderDiameter, 2.0) * PI / 4.0)-
                                    (EXPT(CylinderData.rPistonRodDiameter, 2.0) * PI / 4.0));
    ELSE
        //no special sizes, really use big size
        FCalculateCylinderSize := DINT_TO_REAL(CylinderData.iNumCylinders) *
                                    (EXPT(CylinderData.rCylinderDiameter, 2.0) * PI / 4.0);
    END_IF;
END_IF;

;#END_EDIT_BLOCK END_FUNCTION

#END_OF_IEC_PART

@Puma @IecEditor 6 114 @Pou 25
@@@BEG_Comment@@@
calculate size of cylinder in mm^2
if bSmallSize is TRUE the size only includes the outer ring
@@@END_Comment@@@

@BEG_Contents

@BEG_Func
@RT(17)FuncTreeContainer
0
@END_Func

@BEG_Const
@RT(18)ConstTreeContainer
0
@END_Const

@BEG_Export

@BEG_Kind
@FUNCTION @RT(22)FCalculateCylinderSize @STRUCTURED_TEXT
@RT(4)REAL @RT(0) @RT(0)
@END_Kind

@BEG_Dcl
@RT(16)DclTreeContainer
4
@Var @RT(12)CylinderData @RT(0) @T @T @DERIVED 0 @F @RT(14)tsCylinderData @F
@T
@BEG_Attrib
3 @RT(0) @RT(31)cylinder to calculate size from @RT(0)
@END_Attrib
1 1 @F @F @F @F

@Var @RT(10)bSmallSize @RT(0) @T @F @DT @RT(4)BOOL @RT(0) @T @T @BASIC 0 @F
@F @F
@T
@BEG_Attrib
3 @RT(0) @RT(29)subtract piston rod from size @RT(0)
@END_Attrib
1 1 @F @F @F @F

@Var @RT(18)bCalcHighPressSize @RT(0) @T @F @DT @RT(4)BOOL @RT(0) @T @T @BASIC 0 @F
@F @F
@T
@BEG_Attrib
3 @RT(0) @RT(0) @RT(0)
@END_Attrib
1 1 @F @F @F @F

@Var @RT(2)PI @RT(0) @T @F @DT @RT(4)REAL @RT(0) @T @T @BASIC 0 @F
@F @F
@T
@BEG_Attrib
3 @RT(10)3.14159265 @RT(0) @RT(0)
@END_Attrib
1 15 @F @F @F @F

@END_Dcl

@END_Export

@BEG_Body
@TL(49)
(**************************************** WARNING ********************************************
 *** The KEBA Kemro K2 System including software is not intended for safety control tasks! ***
 ***                       For further information see Comment tab!                        ***
 *********************************************************************************************)

IF CylinderData.rPlungerDiameter <> 0.0 THEN  //plunger available
    IF CylinderData.bMoveWithPlunger THEN //plunger inside highpressure-cylinder -> only used for mold close
        IF bCalcHighPressSize THEN
            FCalculateCylinderSize := DINT_TO_REAL(CylinderData.iNumCylinders) *
                                        ((EXPT(CylinderData.rCylinderDiameter, 2.0) * PI / 4.0)-
                                        (EXPT(CylinderData.rPlungerDiameter, 2.0) * PI / 4.0));
        ELSE
            IF bSmallSize THEN
                FCalculateCylinderSize := DINT_TO_REAL(CylinderData.iNumCylinders) *
                                            ((EXPT(CylinderData.rCylinderDiameter, 2.0) * PI / 4.0)-
                                            (EXPT(CylinderData.rPistonRodDiameter, 2.0) * PI / 4.0));
            ELSE
                FCalculateCylinderSize := DINT_TO_REAL(CylinderData.iNumCylinders) *
                                            (EXPT(CylinderData.rPlungerDiameter, 2.0) * PI / 4.0);
            END_IF;
        END_IF;
    ELSE //plunger used for high pressure build up, differential cylinders used for mold movement
        IF bCalcHighPressSize THEN
            FCalculateCylinderSize := DINT_TO_REAL(CylinderData.iNumCylinders) *
                                        (EXPT(CylinderData.rPlungerDiameter, 2.0) * PI / 4.0);
        ELSE
            IF bSmallSize THEN
                FCalculateCylinderSize := DINT_TO_REAL(CylinderData.iNumCylinders) *
                                            ((EXPT(CylinderData.rCylinderDiameter, 2.0) * PI / 4.0)-
                                            (EXPT(CylinderData.rPistonRodDiameter, 2.0) * PI / 4.0));
            ELSE
                FCalculateCylinderSize := DINT_TO_REAL(CylinderData.iNumCylinders) *
                                            (EXPT(CylinderData.rCylinderDiameter, 2.0) * PI / 4.0);
            END_IF;
        END_IF;
    END_IF;
ELSE //no plunger
    IF bSmallSize THEN
        FCalculateCylinderSize := DINT_TO_REAL(CylinderData.iNumCylinders) *
                                    ((EXPT(CylinderData.rCylinderDiameter, 2.0) * PI / 4.0)-
                                    (EXPT(CylinderData.rPistonRodDiameter, 2.0) * PI / 4.0));
    ELSE
        //no special sizes, really use big size
        FCalculateCylinderSize := DINT_TO_REAL(CylinderData.iNumCylinders) *
                                    (EXPT(CylinderData.rCylinderDiameter, 2.0) * PI / 4.0);
    END_IF;
END_IF;

@END_Body

@END_Contents

(* ---- FCreateIECBaseVersion.pu ---- *)
(*
@h    ! WARNING !
@h    The Kemro K2 system (including software) only meets category B according to EN 954-1,
@h    thus it is not intended for usage in safety-relevant control applications in the field
@h    of personal safety (e.g. emergency stop).
@h    To implement potentially necessary safety-relevant control tasks, always use additional
@h    external safety devices that are intended for the particular purpose, and meet the necessary
@h    functional safety.
@h    For further information see EN 954-1 (EN ISO 13849-1) and/or the K2-x00 user manual, chapter
@h    "CE conformity, directives and standards".

this file is automatically created by clearcase makebaseline
and contains versioninformation of component
*)

IMPORT_OVER_LISTFILE
 FWriteComponentVersion

END_IMPORT

FUNCTION FCreateIECBaseVersion : BOOL #DUMMY_EDIT_BLOCK

VAR CONSTANT
 sComponentName : STRING(255) := 'ApplMoldMachineIECBase';
 iComponentNumber : DINT := 6451;
 sVersionString : STRING(255) := 'ApplMoldMachineIECBase_01.58';
 iVersionMajor : DINT := 1;
 iVersionMinor : DINT := 58;
END_VAR
#BEGIN_EDIT_BLOCK
(**************************************** WARNING ********************************************
 *** The KEBA Kemro K2 System including software is not intended for safety control tasks! ***
 ***                       For further information see Comment tab!                        ***
 *********************************************************************************************)

FCreateIECBaseVersion := FWriteComponentVersion(
        sComponentName,
        iComponentNumber,
        sVersionString,
        iVersionMajor,
        iVersionMinor
);

;#END_EDIT_BLOCK END_FUNCTION

#END_OF_IEC_PART

@Puma @IecEditor 6 68 @Pou 25
@@@BEG_Comment@@@
@h    ! WARNING !
@h    The Kemro K2 system (including software) only meets category B according to EN 954-1,
@h    thus it is not intended for usage in safety-relevant control applications in the field
@h    of personal safety (e.g. emergency stop).
@h    To implement potentially necessary safety-relevant control tasks, always use additional
@h    external safety devices that are intended for the particular purpose, and meet the necessary
@h    functional safety.
@h    For further information see EN 954-1 (EN ISO 13849-1) and/or the K2-x00 user manual, chapter
@h    "CE conformity, directives and standards".

this file is automatically created by clearcase makebaseline
and contains versioninformation of component
@@@END_Comment@@@

@BEG_Contents

@BEG_Func
@RT(17)FuncTreeContainer
1
@Var @RT(22)FWriteComponentVersion @RT(0) @T @F @DT @RT(0) @RT(0) @T @T @UNKNOWN 0 @F
@F @F
@T
@BEG_Attrib
0 @RT(0) @RT(0)
@END_Attrib
1 1 @F @F @F @F

@END_Func

@BEG_Const
@RT(18)ConstTreeContainer
0
@END_Const

@BEG_Export

@BEG_Kind
@FUNCTION @RT(21)FCreateIECBaseVersion @STRUCTURED_TEXT
@RT(4)BOOL @RT(0) @RT(0)
@END_Kind

@BEG_Dcl
@RT(16)DclTreeContainer
5
@Var @RT(14)sComponentName @RT(0) @T @F @DT @RT(11)STRING(255) @RT(0) @T @T @STRING 0 @F @RT(3)255 @F
@F @F
@T
@BEG_Attrib
3 @RT(24)'ApplMoldMachineIECBase' @RT(0) @RT(0)
@END_Attrib
1 15 @F @F @F @F

@Var @RT(16)iComponentNumber @RT(0) @T @F @DT @RT(4)DINT @RT(0) @T @T @BASIC 0 @F
@F @F
@T
@BEG_Attrib
3 @RT(4)6451 @RT(0) @RT(0)
@END_Attrib
1 15 @F @F @F @F

@Var @RT(14)sVersionString @RT(0) @T @F @DT @RT(11)STRING(255) @RT(0) @T @T @STRING 0 @F @RT(3)255 @F
@F @F
@T
@BEG_Attrib
3 @RT(30)'ApplMoldMachineIECBase_01.58' @RT(0) @RT(0)
@END_Attrib
1 15 @F @F @F @F

@Var @RT(13)iVersionMajor @RT(0) @T @F @DT @RT(4)DINT @RT(0) @T @T @BASIC 0 @F
@F @F
@T
@BEG_Attrib
3 @RT(1)1 @RT(0) @RT(0)
@END_Attrib
1 15 @F @F @F @F

@Var @RT(13)iVersionMinor @RT(0) @T @F @DT @RT(4)DINT @RT(0) @T @T @BASIC 0 @F
@F @F
@T
@BEG_Attrib
3 @RT(2)58 @RT(0) @RT(0)
@END_Attrib
1 15 @F @F @F @F

@END_Dcl

@END_Export

@BEG_Body
@TL(13)
(**************************************** WARNING ********************************************
 *** The KEBA Kemro K2 System including software is not intended for safety control tasks! ***
 ***                       For further information see Comment tab!                        ***
 *********************************************************************************************)

FCreateIECBaseVersion := FWriteComponentVersion(
        sComponentName,
        iComponentNumber,
        sVersionString,
        iVersionMajor,
        iVersionMinor
);

@END_Body

@END_Contents

(* ---- FFixCylinderData.pu ---- *)
(*
Fixes wrong values in the CylinderData parameter

Returns TRUE when there was something to fix up
*)

IMPORT_OVER_LISTFILE
 tsCylinderData

END_IMPORT

FUNCTION FFixCylinderData : BOOL #DUMMY_EDIT_BLOCK

VAR_INPUT
 pCylinderData : REFTO tsCylinderData;
END_VAR

VAR
 pCylinderDataTmp : REFTO tsCylinderData;
END_VAR
#BEGIN_EDIT_BLOCK
(**************************************** WARNING ********************************************
 *** The KEBA Kemro K2 System including software is not intended for safety control tasks! ***
 ***                       For further information see Comment tab!                        ***
 *********************************************************************************************)

// to work around can not write to VAR_INPUT
pCylinderDataTmp := pCylinderData;

FFixCylinderData := FALSE;

IF pCylinderDataTmp^.iNumCylinders <= 0 OR pCylinderDataTmp^.iNumCylinders > 9 THEN
   pCylinderDataTmp^.iNumCylinders := 1;
   FFixCylinderData := TRUE;
END_IF;

IF pCylinderDataTmp^.rCylinderDiameter <= 0.0 THEN
   pCylinderDataTmp^.rCylinderDiameter := 20.0;
   FFixCylinderData := TRUE;
END_IF;

//rPistonRodDiameter 0.0 is allowed to have same area on both sides
IF pCylinderDataTmp^.rPistonRodDiameter < 0.0 OR
   pCylinderDataTmp^.rPistonRodDiameter >= pCylinderDataTmp^.rCylinderDiameter THEN
   pCylinderDataTmp^.rPistonRodDiameter := pCylinderDataTmp^.rCylinderDiameter * 0.75;
   FFixCylinderData := TRUE;
END_IF;

;#END_EDIT_BLOCK END_FUNCTION

#END_OF_IEC_PART

@Puma @IecEditor 6 30 @Pou 25
@@@BEG_Comment@@@
Fixes wrong values in the CylinderData parameter

Returns TRUE when there was something to fix up
@@@END_Comment@@@

@BEG_Contents

@BEG_Func
@RT(17)FuncTreeContainer
0
@END_Func

@BEG_Const
@RT(18)ConstTreeContainer
0
@END_Const

@BEG_Export

@BEG_Kind
@FUNCTION @RT(16)FFixCylinderData @STRUCTURED_TEXT
@RT(4)BOOL @RT(0) @RT(0)
@END_Kind

@BEG_Dcl
@RT(16)DclTreeContainer
2
@Var @RT(13)pCylinderData @RT(0) @T @T @REFTO 0 @F @DERIVED 0 @T @T @DT @RT(14)tsCylinderData @RT(0) @T @T @UNKNOWN 0 @F
@F @F
@T
@BEG_Attrib
3 @RT(0) @RT(0) @RT(0)
@END_Attrib
1 1 @F @F @F @F

@Var @RT(16)pCylinderDataTmp @RT(0) @T @T @REFTO 0 @F @DERIVED 0 @T @T @DT @RT(14)tsCylinderData @RT(0) @T @T @UNKNOWN 0 @F
@F @F
@T
@BEG_Attrib
3 @RT(0) @RT(0) @RT(0)
@END_Attrib
1 0 @F @F @F @F

@END_Dcl

@END_Export

@BEG_Body
@TL(30)
(**************************************** WARNING ********************************************
 *** The KEBA Kemro K2 System including software is not intended for safety control tasks! ***
 ***                       For further information see Comment tab!                        ***
 *********************************************************************************************)

// to work around can not write to VAR_INPUT
pCylinderDataTmp := pCylinderData;

FFixCylinderData := FALSE;

IF pCylinderDataTmp^.iNumCylinders <= 0 OR pCylinderDataTmp^.iNumCylinders > 9 THEN
   pCylinderDataTmp^.iNumCylinders := 1;
   FFixCylinderData := TRUE;
END_IF;

IF pCylinderDataTmp^.rCylinderDiameter <= 0.0 THEN
   pCylinderDataTmp^.rCylinderDiameter := 20.0;
   FFixCylinderData := TRUE;
END_IF;

//rPistonRodDiameter 0.0 is allowed to have same area on both sides
IF pCylinderDataTmp^.rPistonRodDiameter < 0.0 OR
   pCylinderDataTmp^.rPistonRodDiameter >= pCylinderDataTmp^.rCylinderDiameter THEN
   pCylinderDataTmp^.rPistonRodDiameter := pCylinderDataTmp^.rCylinderDiameter * 0.75;
   FFixCylinderData := TRUE;
END_IF;

@END_Body

@END_Contents

(* ---- FGetCatConfigValueString.pu ---- *)
(*
@h    ! WARNING !
@h    The Kemro K2 system (including software) only meets category B according to EN 954-1,
@h    thus it is not intended for usage in safety-relevant control applications in the field
@h    of personal safety (e.g. emergency stop).
@h    To implement potentially necessary safety-relevant control tasks, always use additional
@h    external safety devices that are intended for the particular purpose, and meet the necessary
@h    functional safety.
@h    For further information see EN 954-1 (EN ISO 13849-1) and/or the K2-x00 user manual, chapter
@h    "CE conformity, directives and standards".

Function to read a configuration value of type string from uos catalog
*)

IMPORT_OVER_LISTFILE
 KCAT_HandleData
, KCAT_Status

END_IMPORT

FUNCTION FGetCatConfigValueString : STRING(255) #DUMMY_EDIT_BLOCK

VAR_INPUT
 Path : STRING(255) (* node name of config value to read (for example 'KVB_FND.PostScriptDir') *);
 DefaultValue : STRING(255) (* default value is used as return value if status not ok *);
END_VAR

VAR
 DataHandle : KCAT_HandleData;
 sValue : STRING(255);
 Status : KCAT_Status;
END_VAR
#BEGIN_EDIT_BLOCK
(**************************************** WARNING ********************************************
 *** The KEBA Kemro K2 System including software is not intended for safety control tasks! ***
 ***                       For further information see Comment tab!                        ***
 *********************************************************************************************)

    FGetCatConfigValueString := DefaultValue;
    DataHandle := KCAT_GetHandle(Path);
    IF DataHandle.Status = KCAT_Status_OK THEN
        Status := KCAT_GetValue(Handle := DataHandle.Handle,
                                Buffer := sValue);
        IF Status<>KCAT_Status_OK THEN
            RETURN;
        END_IF;

        FGetCatConfigValueString := sValue;
    END_IF;

;#END_EDIT_BLOCK END_FUNCTION

#END_OF_IEC_PART

@Puma @IecEditor 6 68 @Pou 25
@@@BEG_Comment@@@
@h    ! WARNING !
@h    The Kemro K2 system (including software) only meets category B according to EN 954-1,
@h    thus it is not intended for usage in safety-relevant control applications in the field
@h    of personal safety (e.g. emergency stop).
@h    To implement potentially necessary safety-relevant control tasks, always use additional
@h    external safety devices that are intended for the particular purpose, and meet the necessary
@h    functional safety.
@h    For further information see EN 954-1 (EN ISO 13849-1) and/or the K2-x00 user manual, chapter
@h    "CE conformity, directives and standards".

Function to read a configuration value of type string from uos catalog
@@@END_Comment@@@

@BEG_Contents

@BEG_Func
@RT(17)FuncTreeContainer
0
@END_Func

@BEG_Const
@RT(18)ConstTreeContainer
0
@END_Const

@BEG_Export

@BEG_Kind
@FUNCTION @RT(24)FGetCatConfigValueString @STRUCTURED_TEXT
@RT(11)STRING(255) @RT(0) @RT(0)
@END_Kind

@BEG_Dcl
@RT(16)DclTreeContainer
5
@Var @RT(10)DataHandle @RT(0) @T @T @DERIVED 0 @T @T @DT @RT(15)KCAT_HandleData @RT(0) @T @T @UNKNOWN 0 @F
@F @F
@T
@BEG_Attrib
3 @RT(0) @RT(0) @RT(0)
@END_Attrib
1 0 @F @F @F @F

@Var @RT(6)sValue @RT(0) @T @F @DT @RT(11)STRING(255) @RT(0) @T @T @STRING 0 @F @RT(3)255 @F
@F @F
@T
@BEG_Attrib
3 @RT(0) @RT(0) @RT(0)
@END_Attrib
1 0 @F @F @F @F

@Var @RT(6)Status @RT(0) @T @T @DERIVED 0 @T @T @DT @RT(11)KCAT_Status @RT(0) @T @T @UNKNOWN 0 @F
@F @F
@T
@BEG_Attrib
3 @RT(0) @RT(0) @RT(0)
@END_Attrib
1 0 @F @F @F @F

@Var @RT(4)Path @RT(0) @T @F @DT @RT(11)STRING(255) @RT(0) @T @T @STRING 0 @F @RT(3)255 @F
@F @F
@T
@BEG_Attrib
3 @RT(0) @RT(71)node name of config value to read (for example 'KVB_FND.PostScriptDir') @RT(0)
@END_Attrib
1 1 @F @F @F @F

@Var @RT(12)DefaultValue @RT(0) @T @F @DT @RT(11)STRING(255) @RT(0) @T @T @STRING 0 @F @RT(3)255 @F
@F @F
@T
@BEG_Attrib
3 @RT(0) @RT(54)default value is used as return value if status not ok @RT(0)
@END_Attrib
1 1 @F @F @F @F

@END_Dcl

@END_Export

@BEG_Body
@TL(16)
(**************************************** WARNING ********************************************
 *** The KEBA Kemro K2 System including software is not intended for safety control tasks! ***
 ***                       For further information see Comment tab!                        ***
 *********************************************************************************************)

    FGetCatConfigValueString := DefaultValue;
    DataHandle := KCAT_GetHandle(Path);
    IF DataHandle.Status = KCAT_Status_OK THEN
        Status := KCAT_GetValue(Handle := DataHandle.Handle,
                                Buffer := sValue);
        IF Status<>KCAT_Status_OK THEN
            RETURN;
        END_IF;

        FGetCatConfigValueString := sValue;
    END_IF;
@END_Body

@END_Contents

(* ---- FGetHWPath.pu ---- *)
(*
@h    ! WARNING !
@h    The Kemro K2 system (including software) only meets category B according to EN 954-1,
@h    thus it is not intended for usage in safety-relevant control applications in the field
@h    of personal safety (e.g. emergency stop).
@h    To implement potentially necessary safety-relevant control tasks, always use additional
@h    external safety devices that are intended for the particular purpose, and meet the necessary
@h    functional safety.
@h    For further information see EN 954-1 (EN ISO 13849-1) and/or the K2-x00 user manual, chapter
@h    "CE conformity, directives and standards".

This function gets the hardware path for a given endpoint name.
The return value can be simplified by calling the function with bSimplify = TRUE.
Examples:
return value with bSimplify = FALSE:
'IO.ONBOARD.AI:5'
'IO.ONBOARD.KBUS:0.TM240A:4.TI:0'
'IO.ONBOARD.CAN:0.BL210B:1.KBUS:0.AI240A:1.AI:3'

return value with bSimplify = TRUE:
'ONBOARD.AI:5'
'ONBOARD.TM240A:4.TI:0'
'BL210B:1.AI240A:1.AI:3'
*)

IMPORT_OVER_LISTFILE
 FSimplifyHWPath
, KCAT_HandleData
, KCAT_NameData

END_IMPORT

FUNCTION FGetHWPath : STRING(255) #DUMMY_EDIT_BLOCK

VAR_INPUT
 sEndpointName : STRING(255) (* hardware - endpoint  for example: 'FunctionUnit1.ti_2' *);
 bSimplify : BOOL (* TRUE: hardware path will be simplified ('for example 'KBUS:X' is deleted) *);
END_VAR

VAR
 handleData : KCAT_HandleData;
 catNameData : KCAT_NameData;
END_VAR
#BEGIN_EDIT_BLOCK
(**************************************** WARNING ********************************************
 *** The KEBA Kemro K2 System including software is not intended for safety control tasks! ***
 ***                       For further information see Comment tab!                        ***
 *********************************************************************************************)

//get hw path
handleData := KCAT_GetIoHandle(sEndpointName);
catNameData := KCAT_GetName(handleData.Handle);

IF catNameData.Status = KCAT_Status_OK THEN
   IF bSimplify THEN
      FGetHWPath := FSimplifyHWPath(catNameData.Name);
   ELSE
      FGetHWPath := catNameData.Name;
   END_IF;
ELSE
   //return empty string
   FGetHWPath := '';
END_IF;

;#END_EDIT_BLOCK END_FUNCTION

#END_OF_IEC_PART

@Puma @IecEditor 6 120 @Pou 25
@@@BEG_Comment@@@
@h    ! WARNING !
@h    The Kemro K2 system (including software) only meets category B according to EN 954-1,
@h    thus it is not intended for usage in safety-relevant control applications in the field
@h    of personal safety (e.g. emergency stop).
@h    To implement potentially necessary safety-relevant control tasks, always use additional
@h    external safety devices that are intended for the particular purpose, and meet the necessary
@h    functional safety.
@h    For further information see EN 954-1 (EN ISO 13849-1) and/or the K2-x00 user manual, chapter
@h    "CE conformity, directives and standards".

This function gets the hardware path for a given endpoint name.
The return value can be simplified by calling the function with bSimplify = TRUE.
Examples:
return value with bSimplify = FALSE:
'IO.ONBOARD.AI:5'
'IO.ONBOARD.KBUS:0.TM240A:4.TI:0'
'IO.ONBOARD.CAN:0.BL210B:1.KBUS:0.AI240A:1.AI:3'

return value with bSimplify = TRUE:
'ONBOARD.AI:5'
'ONBOARD.TM240A:4.TI:0'
'BL210B:1.AI240A:1.AI:3'
@@@END_Comment@@@

@BEG_Contents

@BEG_Func
@RT(17)FuncTreeContainer
1
@Var @RT(15)FSimplifyHWPath @RT(0) @T @T @DERIVED 0 @F @RT(8)FUNCTION @F
@T
@BEG_Attrib
0 @RT(0) @RT(0)
@END_Attrib
1 1 @F @F @F @F

@END_Func

@BEG_Const
@RT(18)ConstTreeContainer
0
@END_Const

@BEG_Export

@BEG_Kind
@FUNCTION @RT(10)FGetHWPath @STRUCTURED_TEXT
@RT(11)STRING(255) @RT(0) @RT(0)
@END_Kind

@BEG_Dcl
@RT(16)DclTreeContainer
4
@Var @RT(13)sEndpointName @RT(0) @T @F @DT @RT(11)STRING(255) @RT(0) @T @T @STRING 0 @F @RT(3)255 @F
@F @F
@T
@BEG_Attrib
3 @RT(0) @RT(54)hardware - endpoint  for example: 'FunctionUnit1.ti_2' @RT(0)
@END_Attrib
1 1 @F @F @F @F

@Var @RT(10)handleData @RT(0) @T @T @DERIVED 0 @T @T @DT @RT(15)KCAT_HandleData @RT(0) @T @T @UNKNOWN 0 @F
@F @F
@T
@BEG_Attrib
3 @RT(0) @RT(0) @RT(0)
@END_Attrib
1 0 @F @F @F @F

@Var @RT(11)catNameData @RT(0) @T @T @DERIVED 0 @T @T @DT @RT(13)KCAT_NameData @RT(0) @T @T @UNKNOWN 0 @F
@F @F
@T
@BEG_Attrib
3 @RT(0) @RT(0) @RT(0)
@END_Attrib
1 0 @F @F @F @F

@Var @RT(9)bSimplify @RT(0) @T @F @DT @RT(4)BOOL @RT(0) @T @T @BASIC 0 @F
@F @F
@T
@BEG_Attrib
3 @RT(0) @RT(73)TRUE: hardware path will be simplified ('for example 'KBUS:X' is deleted) @RT(0)
@END_Attrib
1 1 @F @F @F @F

@END_Dcl

@END_Export

@BEG_Body
@TL(20)
(**************************************** WARNING ********************************************
 *** The KEBA Kemro K2 System including software is not intended for safety control tasks! ***
 ***                       For further information see Comment tab!                        ***
 *********************************************************************************************)

//get hw path
handleData := KCAT_GetIoHandle(sEndpointName);
catNameData := KCAT_GetName(handleData.Handle);

IF catNameData.Status = KCAT_Status_OK THEN
   IF bSimplify THEN
      FGetHWPath := FSimplifyHWPath(catNameData.Name);
   ELSE
      FGetHWPath := catNameData.Name;
   END_IF;
ELSE
   //return empty string
   FGetHWPath := '';
END_IF;

@END_Body

@END_Contents

(* ---- FReadLineFromFile.pu ---- *)
(*
read one line from a the file File
returns 'EOF_REACHED' at the end of the file
@h WARNING: returns a empty string every second time the function is called
*)

IMPORT_OVER_LISTFILE
 KFILE_Open_Data

END_IMPORT

FUNCTION FReadLineFromFile : STRING(255) #DUMMY_EDIT_BLOCK

VAR_INPUT
 File : KFILE_Open_Data;
END_VAR

VAR
 ReadString : STRING(255) := '';
 DatenLesen : STRING(255);
 readcount : DINT := 0;
END_VAR
#BEGIN_EDIT_BLOCK
REPEAT
    readcount := KFILE_Read(Token:=File.Token,Length:=1,Buffer:=DatenLesen);

    IF readcount<>0
         AND DatenLesen<>'$R'
         AND DatenLesen<>'$N'
         AND DatenLesen<>'$L' THEN
            ReadString := CONCAT(ReadString,DatenLesen);
    END_IF;

UNTIL readcount=0
         OR DatenLesen='$R'
         OR DatenLesen='$N'
         OR DatenLesen='$L'
         OR File.Status = KFILE_Status_NOTOK
END_REPEAT;

IF LEN(ReadString)=0 AND (readcount = 0
    OR File.Status = KFILE_Status_NOTOK) THEN
    ReadString := 'EOF_REACHED';
END_IF;
FReadLineFromFile:=ReadString;

;#END_EDIT_BLOCK END_FUNCTION

#END_OF_IEC_PART

@Puma @IecEditor 6 30 @Pou 25
@@@BEG_Comment@@@
read one line from a the file File
returns 'EOF_REACHED' at the end of the file
@h WARNING: returns a empty string every second time the function is called
@@@END_Comment@@@

@BEG_Contents

@BEG_Func
@RT(17)FuncTreeContainer
0
@END_Func

@BEG_Const
@RT(18)ConstTreeContainer
0
@END_Const

@BEG_Export

@BEG_Kind
@FUNCTION @RT(17)FReadLineFromFile @STRUCTURED_TEXT
@RT(11)STRING(255) @RT(0) @RT(0)
@END_Kind

@BEG_Dcl
@RT(16)DclTreeContainer
4
@Var @RT(4)File @RT(0) @T @T @DERIVED 0 @T @T @DT @RT(15)KFILE_Open_Data @RT(0) @T @T @UNKNOWN 0 @F
@F @F
@T
@BEG_Attrib
3 @RT(0) @RT(0) @RT(0)
@END_Attrib
1 1 @F @F @F @F

@Var @RT(10)ReadString @RT(0) @T @F @DT @RT(11)STRING(255) @RT(0) @T @T @STRING 0 @F @RT(3)255 @F
@F @F
@T
@BEG_Attrib
3 @RT(2)'' @RT(0) @RT(0)
@END_Attrib
1 0 @F @F @F @F

@Var @RT(10)DatenLesen @RT(0) @T @F @DT @RT(11)STRING(255) @RT(0) @T @T @STRING 0 @F @RT(3)255 @F
@F @F
@T
@BEG_Attrib
3 @RT(0) @RT(0) @RT(0)
@END_Attrib
1 0 @F @F @F @F

@Var @RT(9)readcount @RT(0) @T @F @DT @RT(4)DINT @RT(0) @T @T @BASIC 0 @F
@F @F
@T
@BEG_Attrib
3 @RT(1)0 @RT(0) @RT(0)
@END_Attrib
1 0 @F @F @F @F

@END_Dcl

@END_Export

@BEG_Body
@TL(24)
REPEAT
    readcount := KFILE_Read(Token:=File.Token,Length:=1,Buffer:=DatenLesen);

    IF readcount<>0
         AND DatenLesen<>'$R'
         AND DatenLesen<>'$N'
         AND DatenLesen<>'$L' THEN
            ReadString := CONCAT(ReadString,DatenLesen);
    END_IF;

UNTIL readcount=0
         OR DatenLesen='$R'
         OR DatenLesen='$N'
         OR DatenLesen='$L'
         OR File.Status = KFILE_Status_NOTOK
END_REPEAT;

IF LEN(ReadString)=0 AND (readcount = 0
    OR File.Status = KFILE_Status_NOTOK) THEN
    ReadString := 'EOF_REACHED';
END_IF;
FReadLineFromFile:=ReadString;

@END_Body

@END_Contents
